LIN {X 0,Y 487.577,Z 898.273,A -85,B 0,C 180,E1 21910.239,E2 21910.239} C_VEL
LIN {X 0,Y 482.825,Z 918.479,A -85,B 0,C 180,E1 21908.672,E2 21908.672} C_VEL
LIN {X 0,Y 477.745,Z 938.393,A -85,B 0,C 180,E1 21906.843,E2 21906.843} C_VEL
LIN {X 0,Y 473.211,Z 955.74,A -85,B 0,C 180,E1 21905.007,E2 21905.007} C_VEL
LIN {X 0,Y 468.212,Z 974.396,A -85,B 0,C 180,E1 21902.704,E2 21902.704} C_VEL
LIN {X 0,Y 464.166,Z 989.477,A -85,B 0,C 180,E1 21900.556,E2 21900.556} C_VEL
LIN {X 0,Y 459.907,Z 1005.746,A -85,B 0,C 180,E1 21897.868,E2 21897.868} C_VEL
LIN {X 0,Y 456.712,Z 1018.542,A -85,B 0,C 180,E1 21895.411,E2 21895.411} C_VEL
LIN {X 0,Y 453.523,Z 1032.445,A -85,B 0,C 180,E1 21892.285,E2 21892.285} C_VEL
LIN {X 0,Y 451.526,Z 1042.299,A -85,B 0,C 180,E1 21889.67,E2 21889.67} C_VEL
LIN {X 0,Y 449.832,Z 1052.269,A -85,B 0,C 180,E1 21886.53,E2 21886.53} C_VEL
LIN {X 0,Y 448.876,Z 1059.387,A -85,B 0,C 180,E1 21883.781,E2 21883.781} C_VEL
LIN {X 0,Y 448.274,Z 1065.688,A -85,B 0,C 180,E1 21880.799,E2 21880.799} C_VEL
LIN {X 0,Y 447.995,Z 1070.282,A -85,B 0,C 180,E1 21877.825,E2 21877.825} C_VEL
LIN {X 0,Y 447.945,Z 1073.099,A -85,B 0,C 180,E1 21875.251,E2 21875.251} C_VEL
LIN {X 0,Y 447.938,Z 1075.03,A -85,B 0,C 180,E1 21872.303,E2 21872.303} C_VEL
LIN {X 0,Y 447.939,Z 1075.344,A -85,B 0,C 180,E1 21869.361,E2 21869.361} C_VEL
LIN {X 0,Y 447.943,Z 1074.469,A -85,B 0,C 180,E1 21866.801,E2 21866.801} C_VEL
LIN {X 0,Y 447.955,Z 1072.272,A -85,B 0,C 180,E1 21863.978,E2 21863.978} C_VEL
LIN {X 0,Y 448.079,Z 1068.203,A -85,B 0,C 180,E1 21860.884,E2 21860.884} C_VEL
LIN {X 0,Y 448.424,Z 1063.366,A -85,B 0,C 180,E1 21858.204,E2 21858.204} C_VEL
LIN {X 0,Y 449.173,Z 1056.41,A -85,B 0,C 180,E1 21855.167,E2 21855.167} C_VEL
LIN {X 0,Y 450.365,Z 1048.003,A -85,B 0,C 180,E1 21852.262,E2 21852.262} C_VEL
LIN {X 0,Y 452.098,Z 1038.249,A -85,B 0,C 180,E1 21849.411,E2 21849.411} C_VEL
LIN {X 0,Y 454.492,Z 1026.41,A -85,B 0,C 180,E1 21846.534,E2 21846.534} C_VEL
LIN {X 0,Y 457.338,Z 1014.003,A -85,B 0,C 180,E1 21843.931,E2 21843.931} C_VEL
LIN {X 0,Y 461.01,Z 998.825,A -85,B 0,C 180,E1 21841.217,E2 21841.217} C_VEL
LIN {X 0,Y 464.563,Z 984.836,A -85,B 0,C 180,E1 21839.042,E2 21839.042} C_VEL
LIN {X 0,Y 469.251,Z 966.475,A -85,B 0,C 180,E1 21836.577,E2 21836.577} C_VEL
LIN {X 0,Y 473.301,Z 950.565,A -85,B 0,C 180,E1 21834.731,E2 21834.731} C_VEL
LIN {X 0,Y 478.374,Z 930.215,A -85,B 0,C 180,E1 21832.688,E2 21832.688} C_VEL
LIN {X 0,Y 482.676,Z 911.955,A -85,B 0,C 180,E1 21831.121,E2 21831.121} C_VEL
LIN {X 0,Y 487.326,Z 891.147,A -85,B 0,C 180,E1 21829.572,E2 21829.572} C_VEL
LIN {X 0,Y 491.661,Z 869.604,A -85,B 0,C 180,E1 21828.238,E2 21828.238} C_VEL
LIN {X 0,Y 495.61,Z 848.055,A -85,B 0,C 180,E1 21827.107,E2 21827.107} C_VEL
LIN {X 0,Y 499.321,Z 824.384,A -85,B 0,C 180,E1 21826.103,E2 21826.103} C_VEL
LIN {X 0,Y 502.303,Z 802.272,A -85,B 0,C 180,E1 21825.352,E2 21825.352} C_VEL
LIN {X 0,Y 504.984,Z 776.643,A -85,B 0,C 180,E1 21824.697,E2 21824.697} C_VEL
LIN {X 0,Y 506.564,Z 754.118,A -85,B 0,C 180,E1 21824.276,E2 21824.276} C_VEL
LIN {X 0,Y 516.933,Z 505.006,A -85,B 0,C 180,E1 21820.505,E2 21820.505} C_VEL
LIN {X 0,Y 518.425,Z 466.807,A -85,B 0,C 180,E1 21819.907,E2 21819.907} C_VEL
LIN {X 0,Y 506.72,Z 446.358,A -85,B 0,C 180,E1 21817.91,E2 21817.91} C_VEL
LIN {X 0,Y 496.467,Z 429.865,A -85,B 0,C 180,E1 21816.04,E2 21816.04} C_VEL
LIN {X 0,Y 486.048,Z 414.014,A -85,B 0,C 180,E1 21813.99,E2 21813.99} C_VEL
LIN {X 0,Y 476.62,Z 400.744,A -85,B 0,C 180,E1 21811.986,E2 21811.986} C_VEL
LIN {X 0,Y 470.189,Z 391.86,A -85,B 0,C 180,E1 21810.512,E2 21810.512} C_VEL
LIN {X 0,Y 465.532,Z 385.893,A -85,B 0,C 180,E1 21809.392,E2 21809.392} C_VEL
LIN {X 0,Y 461.918,Z 381.059,A -85,B 0,C 180,E1 21808.474,E2 21808.474} C_VEL
LIN {X 0,Y 456.914,Z 374.765,A -85,B 0,C 180,E1 21807.147,E2 21807.147} C_VEL
LIN {X 0,Y 453.412,Z 370.552,A -85,B 0,C 180,E1 21806.171,E2 21806.171} C_VEL
LIN {X 0,Y 451.1,Z 367.867,A -85,B 0,C 180,E1 21805.504,E2 21805.504} C_VEL
LIN {X 0,Y 450.288,Z 365.126,A -85,B 0,C 180,E1 21804.741,E2 21804.741} C_VEL
LIN {X 0,Y 450.26,Z 365.145,A -85,B 0,C 180,E1 21801.142,E2 21801.142} C_VEL
LIN {X 0,Y 450.242,Z 365.132,A -85,B 0,C 180,E1 21797.446,E2 21797.446} C_VEL
LIN {X 0,Y 450.24,Z 365.115,A -85,B 0,C 180,E1 21793.746,E2 21793.746} C_VEL
LIN {X 0,Y 450.274,Z 365.11,A -85,B 0,C 180,E1 21790.233,E2 21790.233} C_VEL
LIN {X 0,Y 450.299,Z 365.136,A -85,B 0,C 180,E1 21786.502,E2 21786.502} C_VEL
LIN {X 0,Y 450.259,Z 365.128,A -85,B 0,C 180,E1 21782.8,E2 21782.8} C_VEL
LIN {X 0,Y 450.236,Z 365.107,A -85,B 0,C 180,E1 21779.237,E2 21779.237} C_VEL
LIN {X 0,Y 450.246,Z 365.129,A -85,B 0,C 180,E1 21775.542,E2 21775.542} C_VEL
LIN {X 0,Y 450.282,Z 365.135,A -85,B 0,C 180,E1 21771.958,E2 21771.958} C_VEL
LIN {X 0,Y 450.284,Z 365.106,A -85,B 0,C 180,E1 21768.212,E2 21768.212} C_VEL
LIN {X 0,Y 450.249,Z 365.117,A -85,B 0,C 180,E1 21764.676,E2 21764.676} C_VEL
LIN {X 0,Y 450.245,Z 365.146,A -85,B 0,C 180,E1 21761.081,E2 21761.081} C_VEL
LIN {X 0,Y 450.26,Z 365.134,A -85,B 0,C 180,E1 21757.407,E2 21757.407} C_VEL
LIN {X 0,Y 450.29,Z 365.115,A -85,B 0,C 180,E1 21753.775,E2 21753.775} C_VEL
LIN {X 0,Y 450.287,Z 365.336,A -85,B 0,C 180,E1 21752.375,E2 21752.375} C_VEL
LIN {X 0,Y 451.296,Z 368.138,A -85,B 0,C 180,E1 21752.02,E2 21752.02} C_VEL
LIN {X 0,Y 453.847,Z 370.847,A -85,B 0,C 180,E1 21751.296,E2 21751.296} C_VEL
LIN {X 0,Y 455.527,Z 371.957,A -85,B 0,C 180,E1 21750.855,E2 21750.855} C_VEL
LIN {X 0,Y 457.684,Z 375.518,A -85,B 0,C 180,E1 21750.233,E2 21750.233} C_VEL
LIN {X 0,Y 460.657,Z 378.21,A -85,B 0,C 180,E1 21749.475,E2 21749.475} C_VEL
LIN {X 0,Y 463.451,Z 382.175,A -85,B 0,C 180,E1 21748.743,E2 21748.743} C_VEL
LIN {X 0,Y 465.734,Z 384.434,A -85,B 0,C 180,E1 21748.192,E2 21748.192} C_VEL
LIN {X 0,Y 469.137,Z 388.783,A -85,B 0,C 180,E1 21747.369,E2 21747.369} C_VEL
LIN {X 0,Y 470.884,Z 390.867,A -85,B 0,C 180,E1 21746.962,E2 21746.962} C_VEL
LIN {X 0,Y 476.097,Z 397.437,A -85,B 0,C 180,E1 21745.783,E2 21745.783} C_VEL
LIN {X 0,Y 480.36,Z 402.894,A -85,B 0,C 180,E1 21744.862,E2 21744.862} C_VEL
LIN {X 0,Y 487.396,Z 412.001,A -85,B 0,C 180,E1 21743.419,E2 21743.419} C_VEL
LIN {X 0,Y 499.444,Z 428.57,A -85,B 0,C 180,E1 21741.124,E2 21741.124} C_VEL
LIN {X 0,Y 511.635,Z 446.615,A -85,B 0,C 180,E1 21738.992,E2 21738.992} C_VEL
LIN {X 0,Y 518.739,Z 458.868,A -85,B 0,C 180,E1 21737.8,E2 21737.8} C_VEL
LIN {X 0,Y 508.149,Z 709.985,A -85,B 0,C 180,E1 21734.008,E2 21734.008} C_VEL
LIN {X 0,Y 506.28,Z 748.548,A -85,B 0,C 180,E1 21733.388,E2 21733.388} C_VEL
LIN {X 0,Y 504.192,Z 772.045,A -85,B 0,C 180,E1 21732.838,E2 21732.838} C_VEL
LIN {X 0,Y 501.494,Z 795.854,A -85,B 0,C 180,E1 21732.105,E2 21732.105} C_VEL
LIN {X 0,Y 498.135,Z 818.964,A -85,B 0,C 180,E1 21731.177,E2 21731.177} C_VEL
LIN {X 0,Y 494.465,Z 841.146,A -85,B 0,C 180,E1 21730.095,E2 21730.095} C_VEL
LIN {X 0,Y 490.296,Z 862.557,A -85,B 0,C 180,E1 21728.827,E2 21728.827} C_VEL
LIN {X 0,Y 486.249,Z 881.746,A -85,B 0,C 180,E1 21727.494,E2 21727.494} C_VEL
LIN {X 0,Y 481.239,Z 903.419,A -85,B 0,C 180,E1 21725.721,E2 21725.721} C_VEL
LIN {X 0,Y 477.113,Z 920.181,A -85,B 0,C 180,E1 21724.126,E2 21724.126} C_VEL
LIN {X 0,Y 472.225,Z 939.257,A -85,B 0,C 180,E1 21722.033,E2 21722.033} C_VEL
LIN {X 0,Y 468.005,Z 955.157,A -85,B 0,C 180,E1 21719.996,E2 21719.996} C_VEL
LIN {X 0,Y 463.735,Z 971.472,A -85,B 0,C 180,E1 21717.602,E2 21717.602} C_VEL
LIN {X 0,Y 459.89,Z 986.038,A -85,B 0,C 180,E1 21715.085,E2 21715.085} C_VEL
LIN {X 0,Y 456.552,Z 999.545,A -85,B 0,C 180,E1 21712.4,E2 21712.4} C_VEL
LIN {X 0,Y 453.842,Z 1010.974,A -85,B 0,C 180,E1 21709.699,E2 21709.699} C_VEL
LIN {X 0,Y 451.777,Z 1020.868,A -85,B 0,C 180,E1 21706.987,E2 21706.987} C_VEL
LIN {X 0,Y 451.27,Z 1023.48,A -85,B 0,C 180,E1 21706.176,E2 21706.176} C_VEL
LIN {X 0,Y 449.761,Z 1026.387,A -85,B 0,C 180,E1 21705.278,E2 21705.278} C_VEL
LIN {X 0,Y 442.431,Z 1033.675,A -85,B 0,C 180,E1 21702.889,E2 21702.889} C_VEL
LIN {X 0,Y 441.394,Z 1035.6,A -85,B 0,C 180,E1 21702.074,E2 21702.074} C_VEL
LIN {X 0,Y 440.648,Z 1041.384,A -85,B 0,C 180,E1 21699.271,E2 21699.271} C_VEL
LIN {X 0,Y 440.168,Z 1046.479,A -85,B 0,C 180,E1 21695.998,E2 21695.998} C_VEL
LIN {X 0,Y 440.009,Z 1049.381,A -85,B 0,C 180,E1 21693.257,E2 21693.257} C_VEL
LIN {X 0,Y 439.954,Z 1051.147,A -85,B 0,C 180,E1 21690.521,E2 21690.521} C_VEL
LIN {X 0,Y 439.94,Z 1051.693,A -85,B 0,C 180,E1 21687.395,E2 21687.395} C_VEL
LIN {X 0,Y 439.969,Z 1050.878,A -85,B 0,C 180,E1 21684.654,E2 21684.654} C_VEL
LIN {X 0,Y 440.043,Z 1049.04,A -85,B 0,C 180,E1 21682.033,E2 21682.033} C_VEL
LIN {X 0,Y 440.31,Z 1045.196,A -85,B 0,C 180,E1 21678.738,E2 21678.738} C_VEL
LIN {X 0,Y 440.816,Z 1040.543,A -85,B 0,C 180,E1 21675.954,E2 21675.954} C_VEL
LIN {X 0,Y 441.744,Z 1034.349,A -85,B 0,C 180,E1 21673.023,E2 21673.023} C_VEL
LIN {X 0,Y 443.258,Z 1026.119,A -85,B 0,C 180,E1 21669.948,E2 21669.948} C_VEL
LIN {X 0,Y 445.115,Z 1017.55,A -85,B 0,C 180,E1 21667.271,E2 21667.271} C_VEL
LIN {X 0,Y 448.164,Z 1005.199,A -85,B 0,C 180,E1 21664.044,E2 21664.044} C_VEL
LIN {X 0,Y 451.208,Z 993.916,A -85,B 0,C 180,E1 21661.546,E2 21661.546} C_VEL
LIN {X 0,Y 455.553,Z 978.507,A -85,B 0,C 180,E1 21658.629,E2 21658.629} C_VEL
LIN {X 0,Y 459.705,Z 964.184,A -85,B 0,C 180,E1 21656.314,E2 21656.314} C_VEL
LIN {X 0,Y 465.039,Z 945.702,A -85,B 0,C 180,E1 21653.752,E2 21653.752} C_VEL
LIN {X 0,Y 469.537,Z 929.823,A -85,B 0,C 180,E1 21651.862,E2 21651.862} C_VEL
LIN {X 0,Y 475.157,Z 909.241,A -85,B 0,C 180,E1 21649.757,E2 21649.757} C_VEL
LIN {X 0,Y 479.806,Z 891.095,A -85,B 0,C 180,E1 21648.175,E2 21648.175} C_VEL
LIN {X 0,Y 484.96,Z 869.463,A -85,B 0,C 180,E1 21646.559,E2 21646.559} C_VEL
LIN {X 0,Y 489.182,Z 849.717,A -85,B 0,C 180,E1 21645.321,E2 21645.321} C_VEL
LIN {X 0,Y 493.411,Z 827.942,A -85,B 0,C 180,E1 21644.162,E2 21644.162} C_VEL
LIN {X 0,Y 497.108,Z 805.082,A -85,B 0,C 180,E1 21643.178,E2 21643.178} C_VEL
LIN {X 0,Y 499.914,Z 784.791,A -85,B 0,C 180,E1 21642.467,E2 21642.467} C_VEL
LIN {X 0,Y 502.662,Z 759.493,A -85,B 0,C 180,E1 21641.784,E2 21641.784} C_VEL
LIN {X 0,Y 504.273,Z 737.798,A -85,B 0,C 180,E1 21641.358,E2 21641.358} C_VEL
LIN {X 0,Y 515.677,Z 490.781,A -85,B 0,C 180,E1 21637.581,E2 21637.581} C_VEL
LIN {X 0,Y 516.812,Z 463.843,A -85,B 0,C 180,E1 21637.148,E2 21637.148} C_VEL
LIN {X 0,Y 508.755,Z 450.942,A -85,B 0,C 180,E1 21635.678,E2 21635.678} C_VEL
LIN {X 0,Y 496.361,Z 433.111,A -85,B 0,C 180,E1 21633.26,E2 21633.26} C_VEL
LIN {X 0,Y 485.835,Z 418.911,A -85,B 0,C 180,E1 21631,E2 21631} C_VEL
LIN {X 0,Y 476.902,Z 407.617,A -85,B 0,C 180,E1 21628.9,E2 21628.9} C_VEL
LIN {X 0,Y 472.696,Z 402.404,A -85,B 0,C 180,E1 21627.837,E2 21627.837} C_VEL
LIN {X 0,Y 468.223,Z 396.919,A -85,B 0,C 180,E1 21626.645,E2 21626.645} C_VEL
LIN {X 0,Y 464.612,Z 392.56,A -85,B 0,C 180,E1 21625.631,E2 21625.631} C_VEL
LIN {X 0,Y 463.434,Z 391.165,A -85,B 0,C 180,E1 21625.29,E2 21625.29} C_VEL
LIN {X 0,Y 460.056,Z 387.445,A -85,B 0,C 180,E1 21624.288,E2 21624.288} C_VEL
LIN {X 0,Y 458.701,Z 385.415,A -85,B 0,C 180,E1 21623.851,E2 21623.851} C_VEL
LIN {X 0,Y 455.354,Z 382.348,A -85,B 0,C 180,E1 21622.803,E2 21622.803} C_VEL
LIN {X 0,Y 453.524,Z 379.251,A -85,B 0,C 180,E1 21622.148,E2 21622.148} C_VEL
LIN {X 0,Y 450.179,Z 376.741,A -85,B 0,C 180,E1 21621.021,E2 21621.021} C_VEL
LIN {X 0,Y 448.267,Z 373.433,A -85,B 0,C 180,E1 21620.261,E2 21620.261} C_VEL
LIN {X 0,Y 447.894,Z 372.768,A -85,B 0,C 180,E1 21620.108,E2 21620.108} C_VEL
LIN {X 0,Y 444.635,Z 370.837,A -85,B 0,C 180,E1 21618.895,E2 21618.895} C_VEL
LIN {X 0,Y 442.875,Z 368.133,A -85,B 0,C 180,E1 21618.12,E2 21618.12} C_VEL
LIN {X 0,Y 442.338,Z 366.106,A -85,B 0,C 180,E1 21617.768,E2 21617.768} C_VEL
LIN {X 0,Y 442.359,Z 366.102,A -85,B 0,C 180,E1 21613.996,E2 21613.996} C_VEL
LIN {X 0,Y 442.321,Z 366.108,A -85,B 0,C 180,E1 21610.287,E2 21610.287} C_VEL
LIN {X 0,Y 442.3,Z 366.118,A -85,B 0,C 180,E1 21606.751,E2 21606.751} C_VEL
LIN {X 0,Y 442.306,Z 366.128,A -85,B 0,C 180,E1 21602.98,E2 21602.98} C_VEL
LIN {X 0,Y 442.335,Z 366.134,A -85,B 0,C 180,E1 21599.352,E2 21599.352} C_VEL
LIN {X 0,Y 442.347,Z 366.12,A -85,B 0,C 180,E1 21595.592,E2 21595.592} C_VEL
LIN {X 0,Y 442.325,Z 366.11,A -85,B 0,C 180,E1 21591.937,E2 21591.937} C_VEL
LIN {X 0,Y 442.302,Z 366.107,A -85,B 0,C 180,E1 21588.261,E2 21588.261} C_VEL
LIN {X 0,Y 442.299,Z 366.106,A -85,B 0,C 180,E1 21584.528,E2 21584.528} C_VEL
LIN {X 0,Y 442.314,Z 366.105,A -85,B 0,C 180,E1 21580.866,E2 21580.866} C_VEL
LIN {X 0,Y 442.322,Z 366.277,A -85,B 0,C 180,E1 21580.516,E2 21580.516} C_VEL
LIN {X 0,Y 443.214,Z 368.939,A -85,B 0,C 180,E1 21580.049,E2 21580.049} C_VEL
LIN {X 0,Y 445.677,Z 371.68,A -85,B 0,C 180,E1 21579.032,E2 21579.032} C_VEL
LIN {X 0,Y 448.061,Z 373.157,A -85,B 0,C 180,E1 21578.154,E2 21578.154} C_VEL
LIN {X 0,Y 450.632,Z 377.217,A -85,B 0,C 180,E1 21577.151,E2 21577.151} C_VEL
LIN {X 0,Y 453.238,Z 379.579,A -85,B 0,C 180,E1 21576.258,E2 21576.258} C_VEL
LIN {X 0,Y 458.645,Z 386.423,A -85,B 0,C 180,E1 21574.462,E2 21574.462} C_VEL
LIN {X 0,Y 461.948,Z 390.347,A -85,B 0,C 180,E1 21573.45,E2 21573.45} C_VEL
LIN {X 0,Y 467.029,Z 396.989,A -85,B 0,C 180,E1 21571.969,E2 21571.969} C_VEL
LIN {X 0,Y 474.172,Z 406.465,A -85,B 0,C 180,E1 21570.05,E2 21570.05} C_VEL
LIN {X 0,Y 482.866,Z 418.454,A -85,B 0,C 180,E1 21567.917,E2 21567.917} C_VEL
LIN {X 0,Y 490.981,Z 430.365,A -85,B 0,C 180,E1 21566.082,E2 21566.082} C_VEL
LIN {X 0,Y 498.672,Z 442.104,A -85,B 0,C 180,E1 21564.463,E2 21564.463} C_VEL
LIN {X 0,Y 508.434,Z 457.967,A -85,B 0,C 180,E1 21562.542,E2 21562.542} C_VEL
LIN {X 0,Y 516.756,Z 472.571,A -85,B 0,C 180,E1 21561.002,E2 21561.002} C_VEL
LIN {X 0,Y 505.459,Z 719.112,A -85,B 0,C 180,E1 21557.239,E2 21557.239} C_VEL
LIN {X 0,Y 503.141,Z 765.997,A -85,B 0,C 180,E1 21556.494,E2 21556.494} C_VEL
LIN {X 0,Y 500.731,Z 790.293,A -85,B 0,C 180,E1 21555.946,E2 21555.946} C_VEL
LIN {X 0,Y 498.012,Z 811.651,A -85,B 0,C 180,E1 21555.318,E2 21555.318} C_VEL
LIN {X 0,Y 494.284,Z 835.385,A -85,B 0,C 180,E1 21554.421,E2 21554.421} C_VEL
LIN {X 0,Y 490.661,Z 855.328,A -85,B 0,C 180,E1 21553.492,E2 21553.492} C_VEL
LIN {X 0,Y 485.976,Z 878.276,A -85,B 0,C 180,E1 21552.209,E2 21552.209} C_VEL
LIN {X 0,Y 481.392,Z 898.253,A -85,B 0,C 180,E1 21550.865,E2 21550.865} C_VEL
LIN {X 0,Y 476.571,Z 918.04,A -85,B 0,C 180,E1 21549.318,E2 21549.318} C_VEL
LIN {X 0,Y 471.365,Z 937.738,A -85,B 0,C 180,E1 21547.5,E2 21547.5} C_VEL
LIN {X 0,Y 466.637,Z 955.097,A -85,B 0,C 180,E1 21545.65,E2 21545.65} C_VEL
LIN {X 0,Y 461.543,Z 973.356,A -85,B 0,C 180,E1 21543.385,E2 21543.385} C_VEL
LIN {X 0,Y 457.296,Z 988.506,A -85,B 0,C 180,E1 21541.212,E2 21541.212} C_VEL
LIN {X 0,Y 452.79,Z 1004.901,A -85,B 0,C 180,E1 21538.489,E2 21538.489} C_VEL
LIN {X 0,Y 449.393,Z 1017.799,A -85,B 0,C 180,E1 21535.987,E2 21535.987} C_VEL
LIN {X 0,Y 446.251,Z 1030.721,A -85,B 0,C 180,E1 21533.086,E2 21533.086} C_VEL
LIN {X 0,Y 443.949,Z 1041.201,A -85,B 0,C 180,E1 21530.295,E2 21530.295} C_VEL
LIN {X 0,Y 442.159,Z 1051.012,A -85,B 0,C 180,E1 21527.232,E2 21527.232} C_VEL
LIN {X 0,Y 440.987,Z 1058.875,A -85,B 0,C 180,E1 21524.175,E2 21524.175} C_VEL
LIN {X 0,Y 440.343,Z 1064.981,A -85,B 0,C 180,E1 21521.261,E2 21521.261} C_VEL
LIN {X 0,Y 440.015,Z 1069.92,A -85,B 0,C 180,E1 21518.099,E2 21518.099} C_VEL
LIN {X 0,Y 439.947,Z 1072.8,A -85,B 0,C 180,E1 21515.455,E2 21515.455} C_VEL
LIN {X 0,Y 439.94,Z 1074.616,A -85,B 0,C 180,E1 21512.736,E2 21512.736} C_VEL
LIN {X 0,Y 439.941,Z 1075.173,A -85,B 0,C 180,E1 21509.609,E2 21509.609} C_VEL
LIN {X 0,Y 439.945,Z 1074.317,A -85,B 0,C 180,E1 21506.873,E2 21506.873} C_VEL
LIN {X 0,Y 439.954,Z 1072.278,A -85,B 0,C 180,E1 21504.13,E2 21504.13} C_VEL
LIN {X 0,Y 440.072,Z 1068.387,A -85,B 0,C 180,E1 21500.98,E2 21500.98} C_VEL
LIN {X 0,Y 440.422,Z 1063.558,A -85,B 0,C 180,E1 21498.21,E2 21498.21} C_VEL
LIN {X 0,Y 441.131,Z 1057.143,A -85,B 0,C 180,E1 21495.294,E2 21495.294} C_VEL
LIN {X 0,Y 442.378,Z 1048.656,A -85,B 0,C 180,E1 21492.234,E2 21492.234} C_VEL
LIN {X 0,Y 444.002,Z 1039.698,A -85,B 0,C 180,E1 21489.527,E2 21489.527} C_VEL
LIN {X 0,Y 446.636,Z 1027.29,A -85,B 0,C 180,E1 21486.376,E2 21486.376} C_VEL
LIN {X 0,Y 449.397,Z 1015.646,A -85,B 0,C 180,E1 21483.862,E2 21483.862} C_VEL
LIN {X 0,Y 453.148,Z 1000.861,A -85,B 0,C 180,E1 21481.103,E2 21481.103} C_VEL
LIN {X 0,Y 456.994,Z 986.23,A -85,B 0,C 180,E1 21478.765,E2 21478.765} C_VEL
LIN {X 0,Y 461.561,Z 969.219,A -85,B 0,C 180,E1 21476.393,E2 21476.393} C_VEL
LIN {X 0,Y 466.175,Z 951.698,A -85,B 0,C 180,E1 21474.309,E2 21474.309} C_VEL
LIN {X 0,Y 471.19,Z 932.534,A -85,B 0,C 180,E1 21472.327,E2 21472.327} C_VEL
LIN {X 0,Y 475.946,Z 913.043,A -85,B 0,C 180,E1 21470.62,E2 21470.62} C_VEL
LIN {X 0,Y 480.325,Z 894.144,A -85,B 0,C 180,E1 21469.182,E2 21469.182} C_VEL
LIN {X 0,Y 485.174,Z 871.29,A -85,B 0,C 180,E1 21467.72,E2 21467.72} C_VEL
LIN {X 0,Y 489.097,Z 850.681,A -85,B 0,C 180,E1 21466.614,E2 21466.614} C_VEL
LIN {X 0,Y 493.184,Z 826.007,A -85,B 0,C 180,E1 21465.533,E2 21465.533} C_VEL
LIN {X 0,Y 496.178,Z 804.692,A -85,B 0,C 180,E1 21464.793,E2 21464.793} C_VEL
LIN {X 0,Y 498.987,Z 779.88,A -85,B 0,C 180,E1 21464.126,E2 21464.126} C_VEL
LIN {X 0,Y 500.74,Z 756.733,A -85,B 0,C 180,E1 21463.676,E2 21463.676} C_VEL
LIN {X 0,Y 511.241,Z 514.011,A -85,B 0,C 180,E1 21459.97,E2 21459.97} C_VEL
LIN {X 0,Y 513.043,Z 470.309,A -85,B 0,C 180,E1 21459.284,E2 21459.284} C_VEL
LIN {X 0,Y 502.048,Z 450.985,A -85,B 0,C 180,E1 21457.351,E2 21457.351} C_VEL
LIN {X 0,Y 490.607,Z 432.404,A -85,B 0,C 180,E1 21455.188,E2 21455.188} C_VEL
LIN {X 0,Y 478.766,Z 414.63,A -85,B 0,C 180,E1 21452.746,E2 21452.746} C_VEL
LIN {X 0,Y 467.489,Z 398.866,A -85,B 0,C 180,E1 21450.174,E2 21450.174} C_VEL
LIN {X 0,Y 458.988,Z 387.726,A -85,B 0,C 180,E1 21448.035,E2 21448.035} C_VEL
LIN {X 0,Y 454.272,Z 381.695,A -85,B 0,C 180,E1 21446.752,E2 21446.752} C_VEL
LIN {X 0,Y 451.019,Z 377.76,A -85,B 0,C 180,E1 21445.826,E2 21445.826} C_VEL
LIN {X 0,Y 448.461,Z 374.594,A -85,B 0,C 180,E1 21445.064,E2 21445.064} C_VEL
LIN {X 0,Y 446.748,Z 372.301,A -85,B 0,C 180,E1 21444.531,E2 21444.531} C_VEL
LIN {X 0,Y 443.911,Z 370.013,A -85,B 0,C 180,E1 21443.672,E2 21443.672} C_VEL
LIN {X 0,Y 442.519,Z 367.142,A -85,B 0,C 180,E1 21443.169,E2 21443.169} C_VEL
LIN {X 0,Y 442.344,Z 366.098,A -85,B 0,C 180,E1 21442.88,E2 21442.88} C_VEL
LIN {X 0,Y 442.308,Z 366.102,A -85,B 0,C 180,E1 21439.272,E2 21439.272} C_VEL
LIN {X 0,Y 442.3,Z 366.115,A -85,B 0,C 180,E1 21435.606,E2 21435.606} C_VEL
LIN {X 0,Y 442.32,Z 366.136,A -85,B 0,C 180,E1 21432.004,E2 21432.004} C_VEL
LIN {X 0,Y 442.348,Z 366.102,A -85,B 0,C 180,E1 21428.318,E2 21428.318} C_VEL
LIN {X 0,Y 442.33,Z 366.094,A -85,B 0,C 180,E1 21424.668,E2 21424.668} C_VEL
LIN {X 0,Y 442.307,Z 366.123,A -85,B 0,C 180,E1 21421.036,E2 21421.036} C_VEL
LIN {X 0,Y 442.302,Z 366.125,A -85,B 0,C 180,E1 21417.279,E2 21417.279} C_VEL
LIN {X 0,Y 442.305,Z 366.098,A -85,B 0,C 180,E1 21413.51,E2 21413.51} C_VEL
LIN {X 0,Y 442.341,Z 366.102,A -85,B 0,C 180,E1 21409.976,E2 21409.976} C_VEL
LIN {X 0,Y 442.36,Z 366.13,A -85,B 0,C 180,E1 21406.137,E2 21406.137} C_VEL
LIN {X 0,Y 442.33,Z 366.113,A -85,B 0,C 180,E1 21402.368,E2 21402.368} C_VEL
LIN {X 0,Y 442.304,Z 366.101,A -85,B 0,C 180,E1 21398.795,E2 21398.795} C_VEL
LIN {X 0,Y 442.305,Z 366.104,A -85,B 0,C 180,E1 21395.028,E2 21395.028} C_VEL
LIN {X 0,Y 442.339,Z 366.294,A -85,B 0,C 180,E1 21394.499,E2 21394.499} C_VEL
LIN {X 0,Y 443.294,Z 369.02,A -85,B 0,C 180,E1 21394.122,E2 21394.122} C_VEL
LIN {X 0,Y 445.743,Z 371.73,A -85,B 0,C 180,E1 21393.343,E2 21393.343} C_VEL
LIN {X 0,Y 447.768,Z 373.027,A -85,B 0,C 180,E1 21392.756,E2 21392.756} C_VEL
LIN {X 0,Y 449.926,Z 376.626,A -85,B 0,C 180,E1 21392.072,E2 21392.072} C_VEL
LIN {X 0,Y 453.113,Z 379.439,A -85,B 0,C 180,E1 21391.185,E2 21391.185} C_VEL
LIN {X 0,Y 455.896,Z 383.357,A -85,B 0,C 180,E1 21390.394,E2 21390.394} C_VEL
LIN {X 0,Y 458.238,Z 385.663,A -85,B 0,C 180,E1 21389.782,E2 21389.782} C_VEL
LIN {X 0,Y 461.633,Z 389.986,A -85,B 0,C 180,E1 21388.896,E2 21388.896} C_VEL
LIN {X 0,Y 463.272,Z 391.839,A -85,B 0,C 180,E1 21388.489,E2 21388.489} C_VEL
LIN {X 0,Y 467.173,Z 396.479,A -85,B 0,C 180,E1 21387.542,E2 21387.542} C_VEL
LIN {X 0,Y 476.963,Z 409.138,A -85,B 0,C 180,E1 21385.308,E2 21385.308} C_VEL
LIN {X 0,Y 484.786,Z 419.482,A -85,B 0,C 180,E1 21383.668,E2 21383.668} C_VEL
LIN {X 0,Y 496.615,Z 435.891,A -85,B 0,C 180,E1 21381.379,E2 21381.379} C_VEL
LIN {X 0,Y 508.771,Z 454.299,A -85,B 0,C 180,E1 21379.215,E2 21379.215} C_VEL
LIN {X 0,Y 513.368,Z 462.385,A -85,B 0,C 180,E1 21378.424,E2 21378.424} C_VEL
LIN {X 0,Y 502.343,Z 714.904,A -85,B 0,C 180,E1 21374.583,E2 21374.583} C_VEL
LIN {X 0,Y 500.516,Z 749.833,A -85,B 0,C 180,E1 21374.008,E2 21374.008} C_VEL
LIN {X 0,Y 498.414,Z 772.695,A -85,B 0,C 180,E1 21373.466,E2 21373.466} C_VEL
LIN {X 0,Y 495.629,Z 796.424,A -85,B 0,C 180,E1 21372.728,E2 21372.728} C_VEL
LIN {X 0,Y 492.352,Z 818.328,A -85,B 0,C 180,E1 21371.846,E2 21371.846} C_VEL
LIN {X 0,Y 488.749,Z 839.499,A -85,B 0,C 180,E1 21370.816,E2 21370.816} C_VEL
LIN {X 0,Y 484.276,Z 862.069,A -85,B 0,C 180,E1 21369.489,E2 21369.489} C_VEL
LIN {X 0,Y 480.234,Z 880.63,A -85,B 0,C 180,E1 21368.198,E2 21368.198} C_VEL
LIN {X 0,Y 475.211,Z 901.882,A -85,B 0,C 180,E1 21366.47,E2 21366.47} C_VEL
LIN {X 0,Y 470.686,Z 919.635,A -85,B 0,C 180,E1 21364.777,E2 21364.777} C_VEL
LIN {X 0,Y 465.808,Z 938.147,A -85,B 0,C 180,E1 21362.747,E2 21362.747} C_VEL
LIN {X 0,Y 461.166,Z 954.845,A -85,B 0,C 180,E1 21360.597,E2 21360.597} C_VEL
LIN {X 0,Y 456.779,Z 970.943,A -85,B 0,C 180,E1 21358.218,E2 21358.218} C_VEL
LIN {X 0,Y 452.707,Z 985.688,A -85,B 0,C 180,E1 21355.652,E2 21355.652} C_VEL
LIN {X 0,Y 449.323,Z 998.642,A -85,B 0,C 180,E1 21353.058,E2 21353.058} C_VEL
LIN {X 0,Y 446.265,Z 1010.913,A -85,B 0,C 180,E1 21350.148,E2 21350.148} C_VEL
LIN {X 0,Y 444.102,Z 1020.716,A -85,B 0,C 180,E1 21347.424,E2 21347.424} C_VEL
LIN {X 0,Y 442.278,Z 1030.14,A -85,B 0,C 180,E1 21344.266,E2 21344.266} C_VEL
LIN {X 0,Y 441.394,Z 1035.6,A -85,B 0,C 180,E1 21342.074,E2 21342.074} C_VEL
LIN {X 0,Y 440.111,Z 1037.86,A -85,B 0,C 180,E1 21341.12,E2 21341.12} C_VEL
LIN {X 0,Y 433.155,Z 1043.266,A -85,B 0,C 180,E1 21338.498,E2 21338.498} C_VEL
LIN {X 0,Y 432.383,Z 1044.478,A -85,B 0,C 180,E1 21337.711,E2 21337.711} C_VEL
LIN {X 0,Y 432.089,Z 1048.284,A -85,B 0,C 180,E1 21334.779,E2 21334.779} C_VEL
LIN {X 0,Y 431.976,Z 1050.837,A -85,B 0,C 180,E1 21331.592,E2 21331.592} C_VEL
LIN {X 0,Y 431.951,Z 1051.8,A -85,B 0,C 180,E1 21328.939,E2 21328.939} C_VEL
LIN {X 0,Y 431.954,Z 1051.698,A -85,B 0,C 180,E1 21326.103,E2 21326.103} C_VEL
LIN {X 0,Y 432.022,Z 1050.014,A -85,B 0,C 180,E1 21322.82,E2 21322.82} C_VEL
LIN {X 0,Y 432.173,Z 1047.424,A -85,B 0,C 180,E1 21320.142,E2 21320.142} C_VEL
LIN {X 0,Y 432.574,Z 1043.346,A -85,B 0,C 180,E1 21317.179,E2 21317.179} C_VEL
LIN {X 0,Y 433.432,Z 1037.204,A -85,B 0,C 180,E1 21313.929,E2 21313.929} C_VEL
LIN {X 0,Y 434.663,Z 1030.406,A -85,B 0,C 180,E1 21311.074,E2 21311.074} C_VEL
LIN {X 0,Y 436.848,Z 1020.417,A -85,B 0,C 180,E1 21307.669,E2 21307.669} C_VEL
LIN {X 0,Y 439.249,Z 1010.8,A -85,B 0,C 180,E1 21304.95,E2 21304.95} C_VEL
LIN {X 0,Y 442.83,Z 997.813,A -85,B 0,C 180,E1 21301.841,E2 21301.841} C_VEL
LIN {X 0,Y 446.49,Z 985.27,A -85,B 0,C 180,E1 21299.297,E2 21299.297} C_VEL
LIN {X 0,Y 451.054,Z 970.157,A -85,B 0,C 180,E1 21296.649,E2 21296.649} C_VEL
LIN {X 0,Y 455.508,Z 955.338,A -85,B 0,C 180,E1 21294.43,E2 21294.43} C_VEL
LIN {X 0,Y 460.715,Z 938.153,A -85,B 0,C 180,E1 21292.185,E2 21292.185} C_VEL
LIN {X 0,Y 465.91,Z 919.972,A -85,B 0,C 180,E1 21290.171,E2 21290.171} C_VEL
LIN {X 0,Y 470.913,Z 901.887,A -85,B 0,C 180,E1 21288.43,E2 21288.43} C_VEL
LIN {X 0,Y 476.312,Z 880.73,A -85,B 0,C 180,E1 21286.703,E2 21286.703} C_VEL
LIN {X 0,Y 480.673,Z 862.161,A -85,B 0,C 180,E1 21285.407,E2 21285.407} C_VEL
LIN {X 0,Y 485.784,Z 837.994,A -85,B 0,C 180,E1 21283.997,E2 21283.997} C_VEL
LIN {X 0,Y 489.516,Z 817.506,A -85,B 0,C 180,E1 21283.008,E2 21283.008} C_VEL
LIN {X 0,Y 493.406,Z 792.396,A -85,B 0,C 180,E1 21282.031,E2 21282.031} C_VEL
LIN {X 0,Y 496.099,Z 770.51,A -85,B 0,C 180,E1 21281.372,E2 21281.372} C_VEL
LIN {X 0,Y 498.452,Z 745.206,A -85,B 0,C 180,E1 21280.804,E2 21280.804} C_VEL
LIN {X 0,Y 501.921,Z 674.53,A -85,B 0,C 180,E1 21279.695,E2 21279.695} C_VEL
LIN {X 0,Y 511.78,Z 467.818,A -85,B 0,C 180,E1 21276.514,E2 21276.514} C_VEL
LIN {X 0,Y 504.78,Z 456.576,A -85,B 0,C 180,E1 21275.2,E2 21275.2} C_VEL
LIN {X 0,Y 492.925,Z 439.35,A -85,B 0,C 180,E1 21272.828,E2 21272.828} C_VEL
LIN {X 0,Y 482.888,Z 425.653,A -85,B 0,C 180,E1 21270.623,E2 21270.623} C_VEL
LIN {X 0,Y 474.182,Z 414.504,A -85,B 0,C 180,E1 21268.53,E2 21268.53} C_VEL
LIN {X 0,Y 470.031,Z 409.325,A -85,B 0,C 180,E1 21267.458,E2 21267.458} C_VEL
LIN {X 0,Y 465.619,Z 403.891,A -85,B 0,C 180,E1 21266.256,E2 21266.256} C_VEL
LIN {X 0,Y 461.89,Z 399.125,A -85,B 0,C 180,E1 21265.175,E2 21265.175} C_VEL
LIN {X 0,Y 457.865,Z 394.726,A -85,B 0,C 180,E1 21263.966,E2 21263.966} C_VEL
LIN {X 0,Y 456.425,Z 392.715,A -85,B 0,C 180,E1 21263.498,E2 21263.498} C_VEL
LIN {X 0,Y 452.979,Z 389.244,A -85,B 0,C 180,E1 21262.382,E2 21262.382} C_VEL
LIN {X 0,Y 451.321,Z 386.663,A -85,B 0,C 180,E1 21261.783,E2 21261.783} C_VEL
LIN {X 0,Y 447.983,Z 383.799,A -85,B 0,C 180,E1 21260.616,E2 21260.616} C_VEL
LIN {X 0,Y 445.946,Z 380.402,A -85,B 0,C 180,E1 21259.79,E2 21259.79} C_VEL
LIN {X 0,Y 442.622,Z 378.058,A -85,B 0,C 180,E1 21258.505,E2 21258.505} C_VEL
LIN {X 0,Y 440.723,Z 374.852,A -85,B 0,C 180,E1 21257.631,E2 21257.631} C_VEL
LIN {X 0,Y 440.365,Z 373.869,A -85,B 0,C 180,E1 21257.441,E2 21257.441} C_VEL
LIN {X 0,Y 437.089,Z 372.153,A -85,B 0,C 180,E1 21256.001,E2 21256.001} C_VEL
LIN {X 0,Y 435.021,Z 369.435,A -85,B 0,C 180,E1 21254.918,E2 21254.918} C_VEL
LIN {X 0,Y 434.375,Z 367.098,A -85,B 0,C 180,E1 21254.463,E2 21254.463} C_VEL
LIN {X 0,Y 434.364,Z 367.103,A -85,B 0,C 180,E1 21250.746,E2 21250.746} C_VEL
LIN {X 0,Y 434.366,Z 367.111,A -85,B 0,C 180,E1 21247.008,E2 21247.008} C_VEL
LIN {X 0,Y 434.383,Z 367.122,A -85,B 0,C 180,E1 21243.299,E2 21243.299} C_VEL
LIN {X 0,Y 434.418,Z 367.114,A -85,B 0,C 180,E1 21239.604,E2 21239.604} C_VEL
LIN {X 0,Y 434.401,Z 367.104,A -85,B 0,C 180,E1 21235.776,E2 21235.776} C_VEL
LIN {X 0,Y 434.377,Z 367.098,A -85,B 0,C 180,E1 21232.061,E2 21232.061} C_VEL
LIN {X 0,Y 434.362,Z 367.095,A -85,B 0,C 180,E1 21228.312,E2 21228.312} C_VEL
LIN {X 0,Y 434.36,Z 367.094,A -85,B 0,C 180,E1 21224.512,E2 21224.512} C_VEL
LIN {X 0,Y 434.417,Z 367.337,A -85,B 0,C 180,E1 21223.829,E2 21223.829} C_VEL
LIN {X 0,Y 435.494,Z 370.263,A -85,B 0,C 180,E1 21223.15,E2 21223.15} C_VEL
LIN {X 0,Y 437.713,Z 372.671,A -85,B 0,C 180,E1 21222.038,E2 21222.038} C_VEL
LIN {X 0,Y 440.378,Z 374.005,A -85,B 0,C 180,E1 21220.881,E2 21220.881} C_VEL
LIN {X 0,Y 442.007,Z 377.269,A -85,B 0,C 180,E1 21220.095,E2 21220.095} C_VEL
LIN {X 0,Y 445.233,Z 380.091,A -85,B 0,C 180,E1 21218.803,E2 21218.803} C_VEL
LIN {X 0,Y 446.288,Z 380.829,A -85,B 0,C 180,E1 21218.409,E2 21218.409} C_VEL
LIN {X 0,Y 448.678,Z 384.586,A -85,B 0,C 180,E1 21217.461,E2 21217.461} C_VEL
LIN {X 0,Y 451.531,Z 387.353,A -85,B 0,C 180,E1 21216.46,E2 21216.46} C_VEL
LIN {X 0,Y 459.737,Z 397.67,A -85,B 0,C 180,E1 21213.765,E2 21213.765} C_VEL
LIN {X 0,Y 464.655,Z 404.165,A -85,B 0,C 180,E1 21212.302,E2 21212.302} C_VEL
LIN {X 0,Y 471.602,Z 413.51,A -85,B 0,C 180,E1 21210.396,E2 21210.396} C_VEL
LIN {X 0,Y 481.089,Z 426.79,A -85,B 0,C 180,E1 21208.03,E2 21208.03} C_VEL
LIN {X 0,Y 492.017,Z 443.215,A -85,B 0,C 180,E1 21205.565,E2 21205.565} C_VEL
LIN {X 0,Y 503.274,Z 461.442,A -85,B 0,C 180,E1 21203.254,E2 21203.254} C_VEL
LIN {X 0,Y 511.643,Z 476.212,A -85,B 0,C 180,E1 21201.651,E2 21201.651} C_VEL
LIN {X 0,Y 499.968,Z 722.479,A -85,B 0,C 180,E1 21197.87,E2 21197.87} C_VEL
LIN {X 0,Y 497.691,Z 766.294,A -85,B 0,C 180,E1 21197.164,E2 21197.164} C_VEL
LIN {X 0,Y 495.246,Z 790.201,A -85,B 0,C 180,E1 21196.621,E2 21196.621} C_VEL
LIN {X 0,Y 492.423,Z 811.739,A -85,B 0,C 180,E1 21195.986,E2 21195.986} C_VEL
LIN {X 0,Y 488.567,Z 835.485,A -85,B 0,C 180,E1 21195.082,E2 21195.082} C_VEL
LIN {X 0,Y 484.947,Z 854.788,A -85,B 0,C 180,E1 21194.179,E2 21194.179} C_VEL
LIN {X 0,Y 480.203,Z 877.436,A -85,B 0,C 180,E1 21192.913,E2 21192.913} C_VEL
LIN {X 0,Y 475.462,Z 897.422,A -85,B 0,C 180,E1 21191.567,E2 21191.567} C_VEL
LIN {X 0,Y 470.467,Z 917.266,A -85,B 0,C 180,E1 21190.009,E2 21190.009} C_VEL
LIN {X 0,Y 464.895,Z 937.64,A -85,B 0,C 180,E1 21188.117,E2 21188.117} C_VEL
LIN {X 0,Y 459.973,Z 955.021,A -85,B 0,C 180,E1 21186.246,E2 21186.246} C_VEL
LIN {X 0,Y 454.665,Z 973.247,A -85,B 0,C 180,E1 21183.958,E2 21183.958} C_VEL
LIN {X 0,Y 450.242,Z 988.386,A -85,B 0,C 180,E1 21181.758,E2 21181.758} C_VEL
LIN {X 0,Y 445.524,Z 1004.762,A -85,B 0,C 180,E1 21178.997,E2 21178.997} C_VEL
LIN {X 0,Y 441.972,Z 1017.607,A -85,B 0,C 180,E1 21176.467,E2 21176.467} C_VEL
LIN {X 0,Y 438.648,Z 1030.56,A -85,B 0,C 180,E1 21173.51,E2 21173.51} C_VEL
LIN {X 0,Y 436.221,Z 1041.033,A -85,B 0,C 180,E1 21170.67,E2 21170.67} C_VEL
LIN {X 0,Y 434.319,Z 1050.833,A -85,B 0,C 180,E1 21167.553,E2 21167.553} C_VEL
LIN {X 0,Y 433.067,Z 1058.69,A -85,B 0,C 180,E1 21164.439,E2 21164.439} C_VEL
LIN {X 0,Y 432.375,Z 1064.792,A -85,B 0,C 180,E1 21161.471,E2 21161.471} C_VEL
LIN {X 0,Y 432.028,Z 1069.722,A -85,B 0,C 180,E1 21158.25,E2 21158.25} C_VEL
LIN {X 0,Y 431.948,Z 1072.642,A -85,B 0,C 180,E1 21155.506,E2 21155.506} C_VEL
LIN {X 0,Y 431.942,Z 1074.478,A -85,B 0,C 180,E1 21152.654,E2 21152.654} C_VEL
LIN {X 0,Y 431.944,Z 1074.935,A -85,B 0,C 180,E1 21149.469,E2 21149.469} C_VEL
LIN {X 0,Y 431.947,Z 1074.097,A -85,B 0,C 180,E1 21146.815,E2 21146.815} C_VEL
LIN {X 0,Y 431.957,Z 1072.052,A -85,B 0,C 180,E1 21144.021,E2 21144.021} C_VEL
LIN {X 0,Y 432.098,Z 1067.939,A -85,B 0,C 180,E1 21140.678,E2 21140.678} C_VEL
LIN {X 0,Y 432.468,Z 1063.258,A -85,B 0,C 180,E1 21137.961,E2 21137.961} C_VEL
LIN {X 0,Y 433.263,Z 1056.581,A -85,B 0,C 180,E1 21134.884,E2 21134.884} C_VEL
LIN {X 0,Y 434.613,Z 1047.978,A -85,B 0,C 180,E1 21131.767,E2 21131.767} C_VEL
LIN {X 0,Y 436.447,Z 1038.639,A -85,B 0,C 180,E1 21128.919,E2 21128.919} C_VEL
LIN {X 0,Y 439.195,Z 1026.418,A -85,B 0,C 180,E1 21125.808,E2 21125.808} C_VEL
LIN {X 0,Y 442.123,Z 1014.703,A -85,B 0,C 180,E1 21123.253,E2 21123.253} C_VEL
LIN {X 0,Y 446.307,Z 998.982,A -85,B 0,C 180,E1 21120.322,E2 21120.322} C_VEL
LIN {X 0,Y 450.249,Z 984.69,A -85,B 0,C 180,E1 21118.031,E2 21118.031} C_VEL
LIN {X 0,Y 455.37,Z 966.303,A -85,B 0,C 180,E1 21115.493,E2 21115.493} C_VEL
LIN {X 0,Y 459.837,Z 950.082,A -85,B 0,C 180,E1 21113.567,E2 21113.567} C_VEL
LIN {X 0,Y 465.189,Z 930.126,A -85,B 0,C 180,E1 21111.519,E2 21111.519} C_VEL
LIN {X 0,Y 469.751,Z 912.077,A -85,B 0,C 180,E1 21109.937,E2 21109.937} C_VEL
LIN {X 0,Y 474.735,Z 891.264,A -85,B 0,C 180,E1 21108.355,E2 21108.355} C_VEL
LIN {X 0,Y 479.385,Z 869.689,A -85,B 0,C 180,E1 21106.996,E2 21106.996} C_VEL
LIN {X 0,Y 483.602,Z 848.094,A -85,B 0,C 180,E1 21105.845,E2 21105.845} C_VEL
LIN {X 0,Y 487.513,Z 824.79,A -85,B 0,C 180,E1 21104.84,E2 21104.84} C_VEL
LIN {X 0,Y 490.647,Z 802.953,A -85,B 0,C 180,E1 21104.086,E2 21104.086} C_VEL
LIN {X 0,Y 493.595,Z 776.73,A -85,B 0,C 180,E1 21103.403,E2 21103.403} C_VEL
LIN {X 0,Y 495.266,Z 754.369,A -85,B 0,C 180,E1 21102.977,E2 21102.977} C_VEL
LIN {X 0,Y 506.399,Z 505.651,A -85,B 0,C 180,E1 21099.158,E2 21099.158} C_VEL
LIN {X 0,Y 507.752,Z 473.861,A -85,B 0,C 180,E1 21098.654,E2 21098.654} C_VEL
LIN {X 0,Y 496.766,Z 454.506,A -85,B 0,C 180,E1 21096.659,E2 21096.659} C_VEL
LIN {X 0,Y 485.526,Z 436.238,A -85,B 0,C 180,E1 21094.459,E2 21094.459} C_VEL
LIN {X 0,Y 474.396,Z 419.479,A -85,B 0,C 180,E1 21092.083,E2 21092.083} C_VEL
LIN {X 0,Y 464.351,Z 405.315,A -85,B 0,C 180,E1 21089.723,E2 21089.723} C_VEL
LIN {X 0,Y 456.195,Z 394.492,A -85,B 0,C 180,E1 21087.618,E2 21087.618} C_VEL
LIN {X 0,Y 451.654,Z 388.602,A -85,B 0,C 180,E1 21086.352,E2 21086.352} C_VEL
LIN {X 0,Y 448.444,Z 384.751,A -85,B 0,C 180,E1 21085.418,E2 21085.418} C_VEL
LIN {X 0,Y 444.619,Z 379.774,A -85,B 0,C 180,E1 21084.231,E2 21084.231} C_VEL
LIN {X 0,Y 441.559,Z 377.023,A -85,B 0,C 180,E1 21083.275,E2 21083.275} C_VEL
LIN {X 0,Y 439.696,Z 373.645,A -85,B 0,C 180,E1 21082.601,E2 21082.601} C_VEL
LIN {X 0,Y 436.563,Z 371.7,A -85,B 0,C 180,E1 21081.568,E2 21081.568} C_VEL
LIN {X 0,Y 434.835,Z 368.902,A -85,B 0,C 180,E1 21080.898,E2 21080.898} C_VEL
LIN {X 0,Y 434.414,Z 367.107,A -85,B 0,C 180,E1 21080.655,E2 21080.655} C_VEL
LIN {X 0,Y 434.406,Z 367.12,A -85,B 0,C 180,E1 21076.759,E2 21076.759} C_VEL
LIN {X 0,Y 434.37,Z 367.098,A -85,B 0,C 180,E1 21073.165,E2 21073.165} C_VEL
LIN {X 0,Y 434.36,Z 367.086,A -85,B 0,C 180,E1 21069.407,E2 21069.407} C_VEL
LIN {X 0,Y 434.362,Z 367.096,A -85,B 0,C 180,E1 21065.548,E2 21065.548} C_VEL
LIN {X 0,Y 434.383,Z 367.125,A -85,B 0,C 180,E1 21061.847,E2 21061.847} C_VEL
LIN {X 0,Y 434.41,Z 367.084,A -85,B 0,C 180,E1 21058.285,E2 21058.285} C_VEL
LIN {X 0,Y 434.396,Z 367.082,A -85,B 0,C 180,E1 21054.452,E2 21054.452} C_VEL
LIN {X 0,Y 434.37,Z 367.117,A -85,B 0,C 180,E1 21050.861,E2 21050.861} C_VEL
LIN {X 0,Y 434.365,Z 367.108,A -85,B 0,C 180,E1 21047.098,E2 21047.098} C_VEL
LIN {X 0,Y 434.373,Z 367.087,A -85,B 0,C 180,E1 21043.415,E2 21043.415} C_VEL
LIN {X 0,Y 434.407,Z 367.088,A -85,B 0,C 180,E1 21039.802,E2 21039.802} C_VEL
LIN {X 0,Y 434.403,Z 367.369,A -85,B 0,C 180,E1 21036.893,E2 21036.893} C_VEL
LIN {X 0,Y 435.405,Z 370.151,A -85,B 0,C 180,E1 21036.448,E2 21036.448} C_VEL
LIN {X 0,Y 438.005,Z 372.837,A -85,B 0,C 180,E1 21035.522,E2 21035.522} C_VEL
LIN {X 0,Y 440.013,Z 374.076,A -85,B 0,C 180,E1 21034.871,E2 21034.871} C_VEL
LIN {X 0,Y 442.037,Z 377.566,A -85,B 0,C 180,E1 21034.151,E2 21034.151} C_VEL
LIN {X 0,Y 445.524,Z 380.607,A -85,B 0,C 180,E1 21033.077,E2 21033.077} C_VEL
LIN {X 0,Y 448.383,Z 384.646,A -85,B 0,C 180,E1 21032.184,E2 21032.184} C_VEL
LIN {X 0,Y 450.75,Z 386.798,A -85,B 0,C 180,E1 21031.515,E2 21031.515} C_VEL
LIN {X 0,Y 454.01,Z 391.044,A -85,B 0,C 180,E1 21030.585,E2 21030.585} C_VEL
LIN {X 0,Y 455.822,Z 392.993,A -85,B 0,C 180,E1 21030.099,E2 21030.099} C_VEL
LIN {X 0,Y 459.596,Z 397.562,A -85,B 0,C 180,E1 21029.107,E2 21029.107} C_VEL
LIN {X 0,Y 465.963,Z 405.657,A -85,B 0,C 180,E1 21027.52,E2 21027.52} C_VEL
LIN {X 0,Y 473.123,Z 414.677,A -85,B 0,C 180,E1 21025.868,E2 21025.868} C_VEL
LIN {X 0,Y 484.592,Z 430.179,A -85,B 0,C 180,E1 21023.43,E2 21023.43} C_VEL
LIN {X 0,Y 496.643,Z 447.502,A -85,B 0,C 180,E1 21021.105,E2 21021.105} C_VEL
LIN {X 0,Y 506.73,Z 463.438,A -85,B 0,C 180,E1 21019.296,E2 21019.296} C_VEL
LIN {X 0,Y 508.051,Z 466.028,A -85,B 0,C 180,E1 21019.058,E2 21019.058} C_VEL
LIN {X 0,Y 496.638,Z 718.586,A -85,B 0,C 180,E1 21015.192,E2 21015.192} C_VEL
LIN {X 0,Y 494.781,Z 751.494,A -85,B 0,C 180,E1 21014.633,E2 21014.633} C_VEL
LIN {X 0,Y 492.67,Z 773.612,A -85,B 0,C 180,E1 21014.101,E2 21014.101} C_VEL
LIN {X 0,Y 489.658,Z 798.079,A -85,B 0,C 180,E1 21013.323,E2 21013.323} C_VEL
LIN {X 0,Y 486.432,Z 818.959,A -85,B 0,C 180,E1 21012.474,E2 21012.474} C_VEL
LIN {X 0,Y 482.523,Z 841.197,A -85,B 0,C 180,E1 21011.379,E2 21011.379} C_VEL
LIN {X 0,Y 478.106,Z 862.578,A -85,B 0,C 180,E1 21010.101,E2 21010.101} C_VEL
LIN {X 0,Y 473.753,Z 881.913,A -85,B 0,C 180,E1 21008.74,E2 21008.74} C_VEL
LIN {X 0,Y 468.395,Z 903.636,A -85,B 0,C 180,E1 21006.936,E2 21006.936} C_VEL
LIN {X 0,Y 463.901,Z 920.654,A -85,B 0,C 180,E1 21005.285,E2 21005.285} C_VEL
LIN {X 0,Y 458.704,Z 939.537,A -85,B 0,C 180,E1 21003.17,E2 21003.17} C_VEL
LIN {X 0,Y 453.988,Z 955.906,A -85,B 0,C 180,E1 21001.022,E2 21001.022} C_VEL
LIN {X 0,Y 449.39,Z 972.081,A -85,B 0,C 180,E1 20998.579,E2 20998.579} C_VEL
LIN {X 0,Y 445.178,Z 986.714,A -85,B 0,C 180,E1 20995.975,E2 20995.975} C_VEL
LIN {X 0,Y 441.519,Z 1000.18,A -85,B 0,C 180,E1 20993.207,E2 20993.207} C_VEL
LIN {X 0,Y 438.535,Z 1011.589,A -85,B 0,C 180,E1 20990.417,E2 20990.417} C_VEL
LIN {X 0,Y 436.196,Z 1021.758,A -85,B 0,C 180,E1 20987.522,E2 20987.522} C_VEL
LIN {X 0,Y 434.361,Z 1030.763,A -85,B 0,C 180,E1 20984.395,E2 20984.395} C_VEL
LIN {X 0,Y 433.253,Z 1037.454,A -85,B 0,C 180,E1 20981.583,E2 20981.583} C_VEL
LIN {X 0,Y 432.461,Z 1043.675,A -85,B 0,C 180,E1 20978.242,E2 20978.242} C_VEL
LIN {X 0,Y 432.383,Z 1044.478,A -85,B 0,C 180,E1 20977.711,E2 20977.711} C_VEL
LIN {X 0,Y 431.252,Z 1046.049,A -85,B 0,C 180,E1 20976.712,E2 20976.712} C_VEL
LIN {X 0,Y 424.68,Z 1049.373,A -85,B 0,C 180,E1 20973.957,E2 20973.957} C_VEL
LIN {X 0,Y 424.015,Z 1050.046,A -85,B 0,C 180,E1 20973.139,E2 20973.139} C_VEL
LIN {X 0,Y 423.97,Z 1051.839,A -85,B 0,C 180,E1 20970,E2 20970} C_VEL
LIN {X 0,Y 423.952,Z 1052.046,A -85,B 0,C 180,E1 20966.89,E2 20966.89} C_VEL
LIN {X 0,Y 423.99,Z 1051.15,A -85,B 0,C 180,E1 20964.18,E2 20964.18} C_VEL
LIN {X 0,Y 424.116,Z 1048.864,A -85,B 0,C 180,E1 20961.048,E2 20961.048} C_VEL
LIN {X 0,Y 424.471,Z 1044.87,A -85,B 0,C 180,E1 20957.846,E2 20957.846} C_VEL
LIN {X 0,Y 425.153,Z 1039.888,A -85,B 0,C 180,E1 20954.867,E2 20954.867} C_VEL
LIN {X 0,Y 426.447,Z 1032.657,A -85,B 0,C 180,E1 20951.547,E2 20951.547} C_VEL
LIN {X 0,Y 428.084,Z 1025.127,A -85,B 0,C 180,E1 20948.743,E2 20948.743} C_VEL
LIN {X 0,Y 430.657,Z 1015.015,A -85,B 0,C 180,E1 20945.589,E2 20945.589} C_VEL
LIN {X 0,Y 433.776,Z 1003.834,A -85,B 0,C 180,E1 20942.696,E2 20942.696} C_VEL
LIN {X 0,Y 437.683,Z 990.946,A -85,B 0,C 180,E1 20939.828,E2 20939.828} C_VEL
LIN {X 0,Y 441.9,Z 977.282,A -85,B 0,C 180,E1 20937.263,E2 20937.263} C_VEL
LIN {X 0,Y 446.55,Z 962.651,A -85,B 0,C 180,E1 20934.868,E2 20934.868} C_VEL
LIN {X 0,Y 451.957,Z 945.292,A -85,B 0,C 180,E1 20932.446,E2 20932.446} C_VEL
LIN {X 0,Y 457.023,Z 928.778,A -85,B 0,C 180,E1 20930.457,E2 20930.457} C_VEL
LIN {X 0,Y 462.732,Z 909.231,A -85,B 0,C 180,E1 20928.442,E2 20928.442} C_VEL
LIN {X 0,Y 467.522,Z 891.777,A -85,B 0,C 180,E1 20926.897,E2 20926.897} C_VEL
LIN {X 0,Y 472.813,Z 871.108,A -85,B 0,C 180,E1 20925.319,E2 20925.319} C_VEL
LIN {X 0,Y 477.553,Z 850.328,A -85,B 0,C 180,E1 20923.996,E2 20923.996} C_VEL
LIN {X 0,Y 481.999,Z 828.767,A -85,B 0,C 180,E1 20922.834,E2 20922.834} C_VEL
LIN {X 0,Y 485.904,Z 806.181,A -85,B 0,C 180,E1 20921.848,E2 20921.848} C_VEL
LIN {X 0,Y 488.82,Z 786.379,A -85,B 0,C 180,E1 20921.143,E2 20921.143} C_VEL
LIN {X 0,Y 491.754,Z 761.454,A -85,B 0,C 180,E1 20920.452,E2 20920.452} C_VEL
LIN {X 0,Y 493.545,Z 739.017,A -85,B 0,C 180,E1 20920.002,E2 20920.002} C_VEL
LIN {X 0,Y 505.626,Z 494.827,A -85,B 0,C 180,E1 20916.221,E2 20916.221} C_VEL
LIN {X 0,Y 506.705,Z 471.513,A -85,B 0,C 180,E1 20915.844,E2 20915.844} C_VEL
LIN {X 0,Y 496.592,Z 455.764,A -85,B 0,C 180,E1 20913.865,E2 20913.865} C_VEL
LIN {X 0,Y 485.373,Z 439.786,A -85,B 0,C 180,E1 20911.482,E2 20911.482} C_VEL
LIN {X 0,Y 475.719,Z 426.782,A -85,B 0,C 180,E1 20909.22,E2 20909.22} C_VEL
LIN {X 0,Y 467.493,Z 416.348,A -85,B 0,C 180,E1 20907.102,E2 20907.102} C_VEL
LIN {X 0,Y 463.038,Z 410.841,A -85,B 0,C 180,E1 20905.862,E2 20905.862} C_VEL
LIN {X 0,Y 458.779,Z 405.565,A -85,B 0,C 180,E1 20904.6,E2 20904.6} C_VEL
LIN {X 0,Y 455.074,Z 401.044,A -85,B 0,C 180,E1 20903.434,E2 20903.434} C_VEL
LIN {X 0,Y 450.464,Z 395.877,A -85,B 0,C 180,E1 20901.895,E2 20901.895} C_VEL
LIN {X 0,Y 449.141,Z 394.029,A -85,B 0,C 180,E1 20901.414,E2 20901.414} C_VEL
LIN {X 0,Y 445.811,Z 390.841,A -85,B 0,C 180,E1 20900.206,E2 20900.206} C_VEL
LIN {X 0,Y 444.018,Z 387.983,A -85,B 0,C 180,E1 20899.468,E2 20899.468} C_VEL
LIN {X 0,Y 440.775,Z 385.427,A -85,B 0,C 180,E1 20898.175,E2 20898.175} C_VEL
LIN {X 0,Y 438.663,Z 381.728,A -85,B 0,C 180,E1 20897.169,E2 20897.169} C_VEL
LIN {X 0,Y 434.968,Z 379.222,A -85,B 0,C 180,E1 20895.466,E2 20895.466} C_VEL
LIN {X 0,Y 433.08,Z 376.196,A -85,B 0,C 180,E1 20894.405,E2 20894.405} C_VEL
LIN {X 0,Y 432.523,Z 374.865,A -85,B 0,C 180,E1 20894.048,E2 20894.048} C_VEL
LIN {X 0,Y 429.116,Z 373.125,A -85,B 0,C 180,E1 20892.105,E2 20892.105} C_VEL
LIN {X 0,Y 427.026,Z 370.28,A -85,B 0,C 180,E1 20890.592,E2 20890.592} C_VEL
LIN {X 0,Y 426.463,Z 368.08,A -85,B 0,C 180,E1 20889.992,E2 20889.992} C_VEL
LIN {X 0,Y 426.437,Z 368.086,A -85,B 0,C 180,E1 20886.327,E2 20886.327} C_VEL
LIN {X 0,Y 426.424,Z 368.095,A -85,B 0,C 180,E1 20882.553,E2 20882.553} C_VEL
LIN {X 0,Y 426.427,Z 368.106,A -85,B 0,C 180,E1 20878.791,E2 20878.791} C_VEL
LIN {X 0,Y 426.437,Z 368.114,A -85,B 0,C 180,E1 20875.023,E2 20875.023} C_VEL
LIN {X 0,Y 426.465,Z 368.095,A -85,B 0,C 180,E1 20871.37,E2 20871.37} C_VEL
LIN {X 0,Y 426.455,Z 368.313,A -85,B 0,C 180,E1 20868.298,E2 20868.298} C_VEL
LIN {X 0,Y 427.411,Z 370.977,A -85,B 0,C 180,E1 20867.434,E2 20867.434} C_VEL
LIN {X 0,Y 429.495,Z 373.449,A -85,B 0,C 180,E1 20865.988,E2 20865.988} C_VEL
LIN {X 0,Y 432.77,Z 375.179,A -85,B 0,C 180,E1 20864.145,E2 20864.145} C_VEL
LIN {X 0,Y 434.443,Z 378.617,A -85,B 0,C 180,E1 20863.142,E2 20863.142} C_VEL
LIN {X 0,Y 437.331,Z 381.042,A -85,B 0,C 180,E1 20861.746,E2 20861.746} C_VEL
LIN {X 0,Y 438.682,Z 381.886,A -85,B 0,C 180,E1 20861.15,E2 20861.15} C_VEL
LIN {X 0,Y 440.746,Z 385.354,A -85,B 0,C 180,E1 20860.174,E2 20860.174} C_VEL
LIN {X 0,Y 444.521,Z 388.609,A -85,B 0,C 180,E1 20858.664,E2 20858.664} C_VEL
LIN {X 0,Y 447.227,Z 392.486,A -85,B 0,C 180,E1 20857.592,E2 20857.592} C_VEL
LIN {X 0,Y 449.677,Z 394.898,A -85,B 0,C 180,E1 20856.719,E2 20856.719} C_VEL
LIN {X 0,Y 457.541,Z 404.981,A -85,B 0,C 180,E1 20854.083,E2 20854.083} C_VEL
LIN {X 0,Y 462.492,Z 411.613,A -85,B 0,C 180,E1 20852.581,E2 20852.581} C_VEL
LIN {X 0,Y 468.947,Z 420.397,A -85,B 0,C 180,E1 20850.773,E2 20850.773} C_VEL
LIN {X 0,Y 478.305,Z 433.707,A -85,B 0,C 180,E1 20848.386,E2 20848.386} C_VEL
LIN {X 0,Y 488.863,Z 449.818,A -85,B 0,C 180,E1 20845.95,E2 20845.95} C_VEL
LIN {X 0,Y 499.986,Z 468.064,A -85,B 0,C 180,E1 20843.615,E2 20843.615} C_VEL
LIN {X 0,Y 506.594,Z 479.918,A -85,B 0,C 180,E1 20842.312,E2 20842.312} C_VEL
LIN {X 0,Y 494.495,Z 726.812,A -85,B 0,C 180,E1 20838.499,E2 20838.499} C_VEL
LIN {X 0,Y 492.31,Z 766.561,A -85,B 0,C 180,E1 20837.85,E2 20837.85} C_VEL
LIN {X 0,Y 489.836,Z 790.096,A -85,B 0,C 180,E1 20837.312,E2 20837.312} C_VEL
LIN {X 0,Y 486.878,Z 812.003,A -85,B 0,C 180,E1 20836.663,E2 20836.663} C_VEL
LIN {X 0,Y 482.863,Z 835.876,A -85,B 0,C 180,E1 20835.745,E2 20835.745} C_VEL
LIN {X 0,Y 479.188,Z 854.851,A -85,B 0,C 180,E1 20834.852,E2 20834.852} C_VEL
LIN {X 0,Y 474.298,Z 877.442,A -85,B 0,C 180,E1 20833.58,E2 20833.58} C_VEL
LIN {X 0,Y 469.42,Z 897.339,A -85,B 0,C 180,E1 20832.231,E2 20832.231} C_VEL
LIN {X 0,Y 464.24,Z 917.229,A -85,B 0,C 180,E1 20830.657,E2 20830.657} C_VEL
LIN {X 0,Y 458.654,Z 936.961,A -85,B 0,C 180,E1 20828.812,E2 20828.812} C_VEL
LIN {X 0,Y 453.696,Z 953.814,A -85,B 0,C 180,E1 20826.989,E2 20826.989} C_VEL
LIN {X 0,Y 447.752,Z 973.418,A -85,B 0,C 180,E1 20824.51,E2 20824.51} C_VEL
LIN {X 0,Y 443.226,Z 988.268,A -85,B 0,C 180,E1 20822.321,E2 20822.321} C_VEL
LIN {X 0,Y 438.297,Z 1004.625,A -85,B 0,C 180,E1 20819.522,E2 20819.522} C_VEL
LIN {X 0,Y 434.57,Z 1017.461,A -85,B 0,C 180,E1 20816.954,E2 20816.954} C_VEL
LIN {X 0,Y 431.071,Z 1030.399,A -85,B 0,C 180,E1 20813.949,E2 20813.949} C_VEL
LIN {X 0,Y 428.483,Z 1040.986,A -85,B 0,C 180,E1 20811.024,E2 20811.024} C_VEL
LIN {X 0,Y 426.465,Z 1050.772,A -85,B 0,C 180,E1 20807.84,E2 20807.84} C_VEL
LIN {X 0,Y 425.154,Z 1058.506,A -85,B 0,C 180,E1 20804.714,E2 20804.714} C_VEL
LIN {X 0,Y 424.411,Z 1064.603,A -85,B 0,C 180,E1 20801.69,E2 20801.69} C_VEL
LIN {X 0,Y 424.042,Z 1069.524,A -85,B 0,C 180,E1 20798.407,E2 20798.407} C_VEL
LIN {X 0,Y 423.95,Z 1072.375,A -85,B 0,C 180,E1 20795.685,E2 20795.685} C_VEL
LIN {X 0,Y 423.945,Z 1074.203,A -85,B 0,C 180,E1 20792.839,E2 20792.839} C_VEL
LIN {X 0,Y 423.947,Z 1074.742,A -85,B 0,C 180,E1 20789.595,E2 20789.595} C_VEL
LIN {X 0,Y 423.949,Z 1073.945,A -85,B 0,C 180,E1 20786.89,E2 20786.89} C_VEL
LIN {X 0,Y 423.955,Z 1072.058,A -85,B 0,C 180,E1 20784.179,E2 20784.179} C_VEL
LIN {X 0,Y 424.076,Z 1068.332,A -85,B 0,C 180,E1 20780.911,E2 20780.911} C_VEL
LIN {X 0,Y 424.478,Z 1063.328,A -85,B 0,C 180,E1 20777.898,E2 20777.898} C_VEL
LIN {X 0,Y 425.217,Z 1057.258,A -85,B 0,C 180,E1 20775.009,E2 20775.009} C_VEL
LIN {X 0,Y 426.677,Z 1048.368,A -85,B 0,C 180,E1 20771.64,E2 20771.64} C_VEL
LIN {X 0,Y 428.526,Z 1039.3,A -85,B 0,C 180,E1 20768.798,E2 20768.798} C_VEL
LIN {X 0,Y 431.5,Z 1026.713,A -85,B 0,C 180,E1 20765.494,E2 20765.494} C_VEL
LIN {X 0,Y 434.54,Z 1015.052,A -85,B 0,C 180,E1 20762.896,E2 20762.896} C_VEL
LIN {X 0,Y 438.889,Z 999.45,A -85,B 0,C 180,E1 20759.92,E2 20759.92} C_VEL
LIN {X 0,Y 443.114,Z 984.724,A -85,B 0,C 180,E1 20757.517,E2 20757.517} C_VEL
LIN {X 0,Y 448.571,Z 965.947,A -85,B 0,C 180,E1 20754.892,E2 20754.892} C_VEL
LIN {X 0,Y 453.173,Z 949.861,A -85,B 0,C 180,E1 20752.961,E2 20752.961} C_VEL
LIN {X 0,Y 458.698,Z 929.968,A -85,B 0,C 180,E1 20750.898,E2 20750.898} C_VEL
LIN {X 0,Y 463.716,Z 910.755,A -85,B 0,C 180,E1 20749.206,E2 20749.206} C_VEL
LIN {X 0,Y 468.837,Z 889.947,A -85,B 0,C 180,E1 20747.629,E2 20747.629} C_VEL
LIN {X 0,Y 473.443,Z 869.222,A -85,B 0,C 180,E1 20746.322,E2 20746.322} C_VEL
LIN {X 0,Y 477.832,Z 847.403,A -85,B 0,C 180,E1 20745.155,E2 20745.155} C_VEL
LIN {X 0,Y 481.835,Z 824.131,A -85,B 0,C 180,E1 20744.152,E2 20744.152} C_VEL
LIN {X 0,Y 485.048,Z 802.306,A -85,B 0,C 180,E1 20743.399,E2 20743.399} C_VEL
LIN {X 0,Y 488.038,Z 776.326,A -85,B 0,C 180,E1 20742.724,E2 20742.724} C_VEL
LIN {X 0,Y 489.749,Z 753.945,A -85,B 0,C 180,E1 20742.296,E2 20742.296} C_VEL
LIN {X 0,Y 501.263,Z 505.468,A -85,B 0,C 180,E1 20738.455,E2 20738.455} C_VEL
LIN {X 0,Y 502.5,Z 477.419,A -85,B 0,C 180,E1 20738.007,E2 20738.007} C_VEL
LIN {X 0,Y 491.324,Z 457.681,A -85,B 0,C 180,E1 20735.907,E2 20735.907} C_VEL
LIN {X 0,Y 480.153,Z 439.521,A -85,B 0,C 180,E1 20733.637,E2 20733.637} C_VEL
LIN {X 0,Y 468.819,Z 422.405,A -85,B 0,C 180,E1 20731.109,E2 20731.109} C_VEL
LIN {X 0,Y 458.193,Z 407.553,A -85,B 0,C 180,E1 20728.478,E2 20728.478} C_VEL
LIN {X 0,Y 449.566,Z 396.077,A -85,B 0,C 180,E1 20726.093,E2 20726.093} C_VEL
LIN {X 0,Y 445.699,Z 391.494,A -85,B 0,C 180,E1 20724.946,E2 20724.946} C_VEL
LIN {X 0,Y 442.505,Z 387.216,A -85,B 0,C 180,E1 20723.929,E2 20723.929} C_VEL
LIN {X 0,Y 439.228,Z 384.03,A -85,B 0,C 180,E1 20722.874,E2 20722.874} C_VEL
LIN {X 0,Y 437.634,Z 381.227,A -85,B 0,C 180,E1 20722.289,E2 20722.289} C_VEL
LIN {X 0,Y 434.401,Z 378.872,A -85,B 0,C 180,E1 20721.185,E2 20721.185} C_VEL
LIN {X 0,Y 432.444,Z 375.567,A -85,B 0,C 180,E1 20720.399,E2 20720.399} C_VEL
LIN {X 0,Y 432.079,Z 374.761,A -85,B 0,C 180,E1 20720.241,E2 20720.241} C_VEL
LIN {X 0,Y 428.916,Z 372.928,A -85,B 0,C 180,E1 20719.049,E2 20719.049} C_VEL
LIN {X 0,Y 426.898,Z 369.924,A -85,B 0,C 180,E1 20718.151,E2 20718.151} C_VEL
LIN {X 0,Y 426.426,Z 368.087,A -85,B 0,C 180,E1 20717.826,E2 20717.826} C_VEL
LIN {X 0,Y 426.442,Z 368.074,A -85,B 0,C 180,E1 20714.114,E2 20714.114} C_VEL
LIN {X 0,Y 426.464,Z 368.076,A -85,B 0,C 180,E1 20710.401,E2 20710.401} C_VEL
LIN {X 0,Y 426.47,Z 368.105,A -85,B 0,C 180,E1 20706.597,E2 20706.597} C_VEL
LIN {X 0,Y 426.446,Z 368.091,A -85,B 0,C 180,E1 20702.756,E2 20702.756} C_VEL
LIN {X 0,Y 426.423,Z 368.071,A -85,B 0,C 180,E1 20699.059,E2 20699.059} C_VEL
LIN {X 0,Y 426.423,Z 368.086,A -85,B 0,C 180,E1 20695.24,E2 20695.24} C_VEL
LIN {X 0,Y 426.434,Z 368.114,A -85,B 0,C 180,E1 20691.505,E2 20691.505} C_VEL
LIN {X 0,Y 426.454,Z 368.076,A -85,B 0,C 180,E1 20687.818,E2 20687.818} C_VEL
LIN {X 0,Y 426.473,Z 368.07,A -85,B 0,C 180,E1 20684.079,E2 20684.079} C_VEL
LIN {X 0,Y 426.458,Z 368.084,A -85,B 0,C 180,E1 20680.267,E2 20680.267} C_VEL
LIN {X 0,Y 426.48,Z 368.249,A -85,B 0,C 180,E1 20679.678,E2 20679.678} C_VEL
LIN {X 0,Y 427.365,Z 370.958,A -85,B 0,C 180,E1 20679.204,E2 20679.204} C_VEL
LIN {X 0,Y 429.721,Z 373.581,A -85,B 0,C 180,E1 20678.215,E2 20678.215} C_VEL
LIN {X 0,Y 432.238,Z 375.085,A -85,B 0,C 180,E1 20677.274,E2 20677.274} C_VEL
LIN {X 0,Y 434.091,Z 378.452,A -85,B 0,C 180,E1 20676.516,E2 20676.516} C_VEL
LIN {X 0,Y 437.283,Z 381.067,A -85,B 0,C 180,E1 20675.407,E2 20675.407} C_VEL
LIN {X 0,Y 437.991,Z 381.856,A -85,B 0,C 180,E1 20675.162,E2 20675.162} C_VEL
LIN {X 0,Y 440.624,Z 385.652,A -85,B 0,C 180,E1 20674.242,E2 20674.242} C_VEL
LIN {X 0,Y 443.311,Z 388.033,A -85,B 0,C 180,E1 20673.402,E2 20673.402} C_VEL
LIN {X 0,Y 446.548,Z 392.308,A -85,B 0,C 180,E1 20672.386,E2 20672.386} C_VEL
LIN {X 0,Y 448.568,Z 394.354,A -85,B 0,C 180,E1 20671.799,E2 20671.799} C_VEL
LIN {X 0,Y 452.237,Z 398.813,A -85,B 0,C 180,E1 20670.749,E2 20670.749} C_VEL
LIN {X 0,Y 458.514,Z 406.657,A -85,B 0,C 180,E1 20669.062,E2 20669.062} C_VEL
LIN {X 0,Y 463.411,Z 412.851,A -85,B 0,C 180,E1 20667.832,E2 20667.832} C_VEL
LIN {X 0,Y 470.492,Z 421.952,A -85,B 0,C 180,E1 20666.165,E2 20666.165} C_VEL
LIN {X 0,Y 481.23,Z 436.582,A -85,B 0,C 180,E1 20663.836,E2 20663.836} C_VEL
LIN {X 0,Y 493.209,Z 454.026,A -85,B 0,C 180,E1 20661.472,E2 20661.472} C_VEL
LIN {X 0,Y 502.801,Z 469.369,A -85,B 0,C 180,E1 20659.713,E2 20659.713} C_VEL
LIN {X 0,Y 491.235,Z 716.868,A -85,B 0,C 180,E1 20655.897,E2 20655.897} C_VEL
LIN {X 0,Y 489.314,Z 750.771,A -85,B 0,C 180,E1 20655.326,E2 20655.326} C_VEL
LIN {X 0,Y 487.1,Z 773.465,A -85,B 0,C 180,E1 20654.781,E2 20654.781} C_VEL
LIN {X 0,Y 484.136,Z 797.158,A -85,B 0,C 180,E1 20654.033,E2 20654.033} C_VEL
LIN {X 0,Y 480.571,Z 819.588,A -85,B 0,C 180,E1 20653.117,E2 20653.117} C_VEL
LIN {X 0,Y 476.548,Z 841.777,A -85,B 0,C 180,E1 20652.015,E2 20652.015} C_VEL
LIN {X 0,Y 471.793,Z 863.976,A -85,B 0,C 180,E1 20650.67,E2 20650.67} C_VEL
LIN {X 0,Y 467.112,Z 884.074,A -85,B 0,C 180,E1 20649.23,E2 20649.23} C_VEL
LIN {X 0,Y 461.787,Z 904.731,A -85,B 0,C 180,E1 20647.477,E2 20647.477} C_VEL
LIN {X 0,Y 457.153,Z 921.671,A -85,B 0,C 180,E1 20645.808,E2 20645.808} C_VEL
LIN {X 0,Y 451.475,Z 941.415,A -85,B 0,C 180,E1 20643.544,E2 20643.544} C_VEL
LIN {X 0,Y 447.009,Z 956.39,A -85,B 0,C 180,E1 20641.543,E2 20641.543} C_VEL
LIN {X 0,Y 442.252,Z 972.428,A -85,B 0,C 180,E1 20639.084,E2 20639.084} C_VEL
LIN {X 0,Y 437.937,Z 986.804,A -85,B 0,C 180,E1 20636.49,E2 20636.49} C_VEL
LIN {X 0,Y 434.034,Z 1000.496,A -85,B 0,C 180,E1 20633.631,E2 20633.631} C_VEL
LIN {X 0,Y 430.845,Z 1012.145,A -85,B 0,C 180,E1 20630.727,E2 20630.727} C_VEL
LIN {X 0,Y 428.321,Z 1022.647,A -85,B 0,C 180,E1 20627.667,E2 20627.667} C_VEL
LIN {X 0,Y 426.445,Z 1031.387,A -85,B 0,C 180,E1 20624.53,E2 20624.53} C_VEL
LIN {X 0,Y 425.213,Z 1038.613,A -85,B 0,C 180,E1 20621.392,E2 20621.392} C_VEL
LIN {X 0,Y 424.455,Z 1044.329,A -85,B 0,C 180,E1 20618.125,E2 20618.125} C_VEL
LIN {X 0,Y 424.131,Z 1048.056,A -85,B 0,C 180,E1 20615.275,E2 20615.275} C_VEL
LIN {X 0,Y 424.015,Z 1050.046,A -85,B 0,C 180,E1 20613.139,E2 20613.139} C_VEL
LIN {X 0,Y 422.997,Z 1050.856,A -85,B 0,C 180,E1 20612.104,E2 20612.104} C_VEL
LIN {X 0,Y 416.589,Z 1052.175,A -85,B 0,C 180,E1 20609.255,E2 20609.255} C_VEL
LIN {X 0,Y 415.945,Z 1052.314,A -85,B 0,C 180,E1 20608.413,E2 20608.413} C_VEL
LIN {X 0,Y 415.972,Z 1051.818,A -85,B 0,C 180,E1 20605.036,E2 20605.036} C_VEL
LIN {X 0,Y 416.052,Z 1050.071,A -85,B 0,C 180,E1 20602.126,E2 20602.126} C_VEL
LIN {X 0,Y 416.291,Z 1047.175,A -85,B 0,C 180,E1 20599.202,E2 20599.202} C_VEL
LIN {X 0,Y 416.939,Z 1042.004,A -85,B 0,C 180,E1 20595.665,E2 20595.665} C_VEL
LIN {X 0,Y 417.92,Z 1036.341,A -85,B 0,C 180,E1 20592.742,E2 20592.742} C_VEL
LIN {X 0,Y 419.71,Z 1028.169,A -85,B 0,C 180,E1 20589.354,E2 20589.354} C_VEL
LIN {X 0,Y 421.935,Z 1019.336,A -85,B 0,C 180,E1 20586.391,E2 20586.391} C_VEL
LIN {X 0,Y 425.07,Z 1008.503,A -85,B 0,C 180,E1 20583.302,E2 20583.302} C_VEL
LIN {X 0,Y 428.861,Z 996.143,A -85,B 0,C 180,E1 20580.378,E2 20580.378} C_VEL
LIN {X 0,Y 433.239,Z 982.686,A -85,B 0,C 180,E1 20577.626,E2 20577.626} C_VEL
LIN {X 0,Y 438.22,Z 967.455,A -85,B 0,C 180,E1 20574.999,E2 20574.999} C_VEL
LIN {X 0,Y 443.075,Z 952.695,A -85,B 0,C 180,E1 20572.786,E2 20572.786} C_VEL
LIN {X 0,Y 449.039,Z 934.034,A -85,B 0,C 180,E1 20570.395,E2 20570.395} C_VEL
LIN {X 0,Y 454.325,Z 916.902,A -85,B 0,C 180,E1 20568.513,E2 20568.513} C_VEL
LIN {X 0,Y 460.35,Z 896.166,A -85,B 0,C 180,E1 20566.572,E2 20566.572} C_VEL
LIN {X 0,Y 465.245,Z 877.922,A -85,B 0,C 180,E1 20565.116,E2 20565.116} C_VEL
LIN {X 0,Y 470.527,Z 856.532,A -85,B 0,C 180,E1 20563.658,E2 20563.658} C_VEL
LIN {X 0,Y 475.1,Z 835.421,A -85,B 0,C 180,E1 20562.468,E2 20562.468} C_VEL
LIN {X 0,Y 479.346,Z 813.232,A -85,B 0,C 180,E1 20561.418,E2 20561.418} C_VEL
LIN {X 0,Y 482.959,Z 790.065,A -85,B 0,C 180,E1 20560.552,E2 20560.552} C_VEL
LIN {X 0,Y 485.748,Z 768.223,A -85,B 0,C 180,E1 20559.906,E2 20559.906} C_VEL
LIN {X 0,Y 488.106,Z 742.445,A -85,B 0,C 180,E1 20559.351,E2 20559.351} C_VEL
LIN {X 0,Y 500.072,Z 508.874,A -85,B 0,C 180,E1 20555.706,E2 20555.706} C_VEL
LIN {X 0,Y 501.723,Z 475.289,A -85,B 0,C 180,E1 20555.167,E2 20555.167} C_VEL
LIN {X 0,Y 491.043,Z 458.951,A -85,B 0,C 180,E1 20553.004,E2 20553.004} C_VEL
LIN {X 0,Y 480.225,Z 443.43,A -85,B 0,C 180,E1 20550.603,E2 20550.603} C_VEL
LIN {X 0,Y 469.661,Z 429.257,A -85,B 0,C 180,E1 20547.998,E2 20547.998} C_VEL
LIN {X 0,Y 460.98,Z 418.3,A -85,B 0,C 180,E1 20545.606,E2 20545.606} C_VEL
LIN {X 0,Y 456.288,Z 412.56,A -85,B 0,C 180,E1 20544.191,E2 20544.191} C_VEL
LIN {X 0,Y 451.936,Z 407.223,A -85,B 0,C 180,E1 20542.779,E2 20542.779} C_VEL
LIN {X 0,Y 448.305,Z 403.012,A -85,B 0,C 180,E1 20541.525,E2 20541.525} C_VEL
LIN {X 0,Y 447.158,Z 401.478,A -85,B 0,C 180,E1 20541.101,E2 20541.101} C_VEL
LIN {X 0,Y 443.662,Z 397.874,A -85,B 0,C 180,E1 20539.793,E2 20539.793} C_VEL
LIN {X 0,Y 442.109,Z 395.52,A -85,B 0,C 180,E1 20539.144,E2 20539.144} C_VEL
LIN {X 0,Y 438.805,Z 392.613,A -85,B 0,C 180,E1 20537.779,E2 20537.779} C_VEL
LIN {X 0,Y 436.709,Z 389.232,A -85,B 0,C 180,E1 20536.768,E2 20536.768} C_VEL
LIN {X 0,Y 433.255,Z 386.635,A -85,B 0,C 180,E1 20535.117,E2 20535.117} C_VEL
LIN {X 0,Y 431.273,Z 383.204,A -85,B 0,C 180,E1 20533.953,E2 20533.953} C_VEL
LIN {X 0,Y 430.836,Z 382.617,A -85,B 0,C 180,E1 20533.693,E2 20533.693} C_VEL
LIN {X 0,Y 427.55,Z 380.636,A -85,B 0,C 180,E1 20531.74,E2 20531.74} C_VEL
LIN {X 0,Y 425.626,Z 377.822,A -85,B 0,C 180,E1 20530.285,E2 20530.285} C_VEL
LIN {X 0,Y 424.917,Z 375.931,A -85,B 0,C 180,E1 20529.618,E2 20529.618} C_VEL
LIN {X 0,Y 420.979,Z 373.898,A -85,B 0,C 180,E1 20525.862,E2 20525.862} C_VEL
LIN {X 0,Y 418.688,Z 370.127,A -85,B 0,C 180,E1 20520.547,E2 20520.547} C_VEL
LIN {X 0,Y 418.612,Z 369.749,A -85,B 0,C 180,E1 20519.179,E2 20519.179} C_VEL
LIN {X 0,Y 418.818,Z 370.545,A -85,B 0,C 180,E1 20516.989,E2 20516.989} C_VEL
LIN {X 0,Y 423.403,Z 375.494,A -85,B 0,C 180,E1 20509.936,E2 20509.936} C_VEL
LIN {X 0,Y 425.089,Z 376.181,A -85,B 0,C 180,E1 20508.57,E2 20508.57} C_VEL
LIN {X 0,Y 426.592,Z 379.531,A -85,B 0,C 180,E1 20507.272,E2 20507.272} C_VEL
LIN {X 0,Y 429.411,Z 381.997,A -85,B 0,C 180,E1 20505.435,E2 20505.435} C_VEL
LIN {X 0,Y 431.26,Z 383.048,A -85,B 0,C 180,E1 20504.398,E2 20504.398} C_VEL
LIN {X 0,Y 433.226,Z 386.626,A -85,B 0,C 180,E1 20503.232,E2 20503.232} C_VEL
LIN {X 0,Y 436.396,Z 389.06,A -85,B 0,C 180,E1 20501.705,E2 20501.705} C_VEL
LIN {X 0,Y 437.075,Z 389.746,A -85,B 0,C 180,E1 20501.389,E2 20501.389} C_VEL
LIN {X 0,Y 439.638,Z 393.534,A -85,B 0,C 180,E1 20500.191,E2 20500.191} C_VEL
LIN {X 0,Y 442.695,Z 396.176,A -85,B 0,C 180,E1 20498.953,E2 20498.953} C_VEL
LIN {X 0,Y 445.617,Z 400.199,A -85,B 0,C 180,E1 20497.785,E2 20497.785} C_VEL
LIN {X 0,Y 448.034,Z 402.698,A -85,B 0,C 180,E1 20496.907,E2 20496.907} C_VEL
LIN {X 0,Y 455.36,Z 412.285,A -85,B 0,C 180,E1 20494.404,E2 20494.404} C_VEL
LIN {X 0,Y 460.534,Z 419.318,A -85,B 0,C 180,E1 20492.804,E2 20492.804} C_VEL
LIN {X 0,Y 466.618,Z 427.734,A -85,B 0,C 180,E1 20491.069,E2 20491.069} C_VEL
LIN {X 0,Y 475.649,Z 440.785,A -85,B 0,C 180,E1 20488.719,E2 20488.719} C_VEL
LIN {X 0,Y 485.731,Z 456.417,A -85,B 0,C 180,E1 20486.34,E2 20486.34} C_VEL
LIN {X 0,Y 496.408,Z 474.181,A -85,B 0,C 180,E1 20484.044,E2 20484.044} C_VEL
LIN {X 0,Y 501.607,Z 483.771,A -85,B 0,C 180,E1 20482.984,E2 20482.984} C_VEL
LIN {X 0,Y 489.101,Z 730.776,A -85,B 0,C 180,E1 20479.148,E2 20479.148} C_VEL
LIN {X 0,Y 486.969,Z 767.159,A -85,B 0,C 180,E1 20478.543,E2 20478.543} C_VEL
LIN {X 0,Y 484.48,Z 790.135,A -85,B 0,C 180,E1 20478.015,E2 20478.015} C_VEL
LIN {X 0,Y 481.317,Z 812.88,A -85,B 0,C 180,E1 20477.336,E2 20477.336} C_VEL
LIN {X 0,Y 477.335,Z 835.692,A -85,B 0,C 180,E1 20476.45,E2 20476.45} C_VEL
LIN {X 0,Y 473.495,Z 854.917,A -85,B 0,C 180,E1 20475.542,E2 20475.542} C_VEL
LIN {X 0,Y 468.282,Z 878.153,A -85,B 0,C 180,E1 20474.218,E2 20474.218} C_VEL
LIN {X 0,Y 463.407,Z 897.39,A -85,B 0,C 180,E1 20472.902,E2 20472.902} C_VEL
LIN {X 0,Y 457.88,Z 917.929,A -85,B 0,C 180,E1 20471.261,E2 20471.261} C_VEL
LIN {X 0,Y 451.979,Z 937.935,A -85,B 0,C 180,E1 20469.355,E2 20469.355} C_VEL
LIN {X 0,Y 446.652,Z 955.402,A -85,B 0,C 180,E1 20467.43,E2 20467.43} C_VEL
LIN {X 0,Y 441.063,Z 973.032,A -85,B 0,C 180,E1 20465.157,E2 20465.157} C_VEL
LIN {X 0,Y 436.255,Z 988.151,A -85,B 0,C 180,E1 20462.902,E2 20462.902} C_VEL
LIN {X 0,Y 431.109,Z 1004.489,A -85,B 0,C 180,E1 20460.065,E2 20460.065} C_VEL
LIN {X 0,Y 427.269,Z 1017.077,A -85,B 0,C 180,E1 20457.509,E2 20457.509} C_VEL
LIN {X 0,Y 423.524,Z 1030.24,A -85,B 0,C 180,E1 20454.403,E2 20454.403} C_VEL
LIN {X 0,Y 420.817,Z 1040.699,A -85,B 0,C 180,E1 20451.464,E2 20451.464} C_VEL
LIN {X 0,Y 418.67,Z 1050.475,A -85,B 0,C 180,E1 20448.232,E2 20448.232} C_VEL
LIN {X 0,Y 417.246,Z 1058.322,A -85,B 0,C 180,E1 20445,E2 20445} C_VEL
LIN {X 0,Y 416.452,Z 1064.415,A -85,B 0,C 180,E1 20441.916,E2 20441.916} C_VEL
LIN {X 0,Y 416.053,Z 1069.326,A -85,B 0,C 180,E1 20438.569,E2 20438.569} C_VEL
LIN {X 0,Y 415.953,Z 1072.173,A -85,B 0,C 180,E1 20435.795,E2 20435.795} C_VEL
LIN {X 0,Y 415.947,Z 1073.996,A -85,B 0,C 180,E1 20432.894,E2 20432.894} C_VEL
LIN {X 0,Y 415.951,Z 1074.526,A -85,B 0,C 180,E1 20429.587,E2 20429.587} C_VEL
LIN {X 0,Y 415.951,Z 1073.724,A -85,B 0,C 180,E1 20426.831,E2 20426.831} C_VEL
LIN {X 0,Y 415.958,Z 1071.831,A -85,B 0,C 180,E1 20424.067,E2 20424.067} C_VEL
LIN {X 0,Y 416.09,Z 1068.093,A -85,B 0,C 180,E1 20420.735,E2 20420.735} C_VEL
LIN {X 0,Y 416.522,Z 1063.082,A -85,B 0,C 180,E1 20417.664,E2 20417.664} C_VEL
LIN {X 0,Y 417.312,Z 1057.005,A -85,B 0,C 180,E1 20414.718,E2 20414.718} C_VEL
LIN {X 0,Y 418.828,Z 1048.271,A -85,B 0,C 180,E1 20411.343,E2 20411.343} C_VEL
LIN {X 0,Y 420.717,Z 1039.492,A -85,B 0,C 180,E1 20408.531,E2 20408.531} C_VEL
LIN {X 0,Y 423.668,Z 1027.59,A -85,B 0,C 180,E1 20405.308,E2 20405.308} C_VEL
LIN {X 0,Y 426.974,Z 1015.4,A -85,B 0,C 180,E1 20402.527,E2 20402.527} C_VEL
LIN {X 0,Y 431.27,Z 1000.7,A -85,B 0,C 180,E1 20399.64,E2 20399.64} C_VEL
LIN {X 0,Y 435.756,Z 985.622,A -85,B 0,C 180,E1 20397.122,E2 20397.122} C_VEL
LIN {X 0,Y 440.916,Z 968.695,A -85,B 0,C 180,E1 20394.671,E2 20394.671} C_VEL
LIN {X 0,Y 446.124,Z 951.105,A -85,B 0,C 180,E1 20392.506,E2 20392.506} C_VEL
LIN {X 0,Y 451.673,Z 932.049,A -85,B 0,C 180,E1 20390.472,E2 20390.472} C_VEL
LIN {X 0,Y 457.131,Z 911.839,A -85,B 0,C 180,E1 20388.657,E2 20388.657} C_VEL
LIN {X 0,Y 462.399,Z 891.244,A -85,B 0,C 180,E1 20387.066,E2 20387.066} C_VEL
LIN {X 0,Y 467.35,Z 869.768,A -85,B 0,C 180,E1 20385.69,E2 20385.69} C_VEL
LIN {X 0,Y 471.676,Z 848.949,A -85,B 0,C 180,E1 20384.562,E2 20384.562} C_VEL
LIN {X 0,Y 476.012,Z 824.836,A -85,B 0,C 180,E1 20383.501,E2 20383.501} C_VEL
LIN {X 0,Y 479.336,Z 802.967,A -85,B 0,C 180,E1 20382.738,E2 20382.738} C_VEL
LIN {X 0,Y 482.499,Z 776.475,A -85,B 0,C 180,E1 20382.041,E2 20382.041} C_VEL
LIN {X 0,Y 484.261,Z 754.165,A -85,B 0,C 180,E1 20381.611,E2 20381.611} C_VEL
LIN {X 0,Y 496.168,Z 506.014,A -85,B 0,C 180,E1 20377.749,E2 20377.749} C_VEL
LIN {X 0,Y 497.264,Z 480.875,A -85,B 0,C 180,E1 20377.337,E2 20377.337} C_VEL
LIN {X 0,Y 485.976,Z 460.861,A -85,B 0,C 180,E1 20375.141,E2 20375.141} C_VEL
LIN {X 0,Y 475.949,Z 444.657,A -85,B 0,C 180,E1 20373.036,E2 20373.036} C_VEL
LIN {X 0,Y 465.74,Z 428.971,A -85,B 0,C 180,E1 20370.692,E2 20370.692} C_VEL
LIN {X 0,Y 455.376,Z 414.304,A -85,B 0,C 180,E1 20368.063,E2 20368.063} C_VEL
LIN {X 0,Y 446.885,Z 402.869,A -85,B 0,C 180,E1 20365.655,E2 20365.655} C_VEL
LIN {X 0,Y 440.971,Z 395.228,A -85,B 0,C 180,E1 20363.804,E2 20363.804} C_VEL
LIN {X 0,Y 436.919,Z 391.036,A -85,B 0,C 180,E1 20362.469,E2 20362.469} C_VEL
LIN {X 0,Y 435.592,Z 388.754,A -85,B 0,C 180,E1 20361.973,E2 20361.973} C_VEL
LIN {X 0,Y 432.26,Z 386.031,A -85,B 0,C 180,E1 20360.798,E2 20360.798} C_VEL
LIN {X 0,Y 429.94,Z 382.324,A -85,B 0,C 180,E1 20359.849,E2 20359.849} C_VEL
LIN {X 0,Y 426.729,Z 379.982,A -85,B 0,C 180,E1 20358.583,E2 20358.583} C_VEL
LIN {X 0,Y 424.725,Z 376.641,A -85,B 0,C 180,E1 20357.644,E2 20357.644} C_VEL
LIN {X 0,Y 424.263,Z 375.798,A -85,B 0,C 180,E1 20357.416,E2 20357.416} C_VEL
LIN {X 0,Y 420.826,Z 373.806,A -85,B 0,C 180,E1 20355.857,E2 20355.857} C_VEL
LIN {X 0,Y 419.073,Z 371.165,A -85,B 0,C 180,E1 20354.897,E2 20354.897} C_VEL
LIN {X 0,Y 418.534,Z 369.058,A -85,B 0,C 180,E1 20354.461,E2 20354.461} C_VEL
LIN {X 0,Y 418.524,Z 369.067,A -85,B 0,C 180,E1 20350.601,E2 20350.601} C_VEL
LIN {X 0,Y 418.506,Z 369.102,A -85,B 0,C 180,E1 20346.861,E2 20346.861} C_VEL
LIN {X 0,Y 418.486,Z 369.072,A -85,B 0,C 180,E1 20343.15,E2 20343.15} C_VEL
LIN {X 0,Y 418.483,Z 369.059,A -85,B 0,C 180,E1 20339.315,E2 20339.315} C_VEL
LIN {X 0,Y 418.489,Z 369.078,A -85,B 0,C 180,E1 20335.478,E2 20335.478} C_VEL
LIN {X 0,Y 418.51,Z 369.095,A -85,B 0,C 180,E1 20331.758,E2 20331.758} C_VEL
LIN {X 0,Y 418.525,Z 369.06,A -85,B 0,C 180,E1 20328.004,E2 20328.004} C_VEL
LIN {X 0,Y 418.516,Z 369.061,A -85,B 0,C 180,E1 20324.327,E2 20324.327} C_VEL
LIN {X 0,Y 418.514,Z 369.269,A -85,B 0,C 180,E1 20323.071,E2 20323.071} C_VEL
LIN {X 0,Y 419.428,Z 371.93,A -85,B 0,C 180,E1 20322.473,E2 20322.473} C_VEL
LIN {X 0,Y 421.919,Z 374.717,A -85,B 0,C 180,E1 20321.198,E2 20321.198} C_VEL
LIN {X 0,Y 424.495,Z 375.974,A -85,B 0,C 180,E1 20320.065,E2 20320.065} C_VEL
LIN {X 0,Y 426.155,Z 379.317,A -85,B 0,C 180,E1 20319.25,E2 20319.25} C_VEL
LIN {X 0,Y 428.96,Z 381.799,A -85,B 0,C 180,E1 20318.102,E2 20318.102} C_VEL
LIN {X 0,Y 430.281,Z 382.728,A -85,B 0,C 180,E1 20317.598,E2 20317.598} C_VEL
LIN {X 0,Y 432.629,Z 386.398,A -85,B 0,C 180,E1 20316.648,E2 20316.648} C_VEL
LIN {X 0,Y 435.876,Z 389.234,A -85,B 0,C 180,E1 20315.503,E2 20315.503} C_VEL
LIN {X 0,Y 438.94,Z 393.394,A -85,B 0,C 180,E1 20314.426,E2 20314.426} C_VEL
LIN {X 0,Y 441.207,Z 395.549,A -85,B 0,C 180,E1 20313.701,E2 20313.701} C_VEL
LIN {X 0,Y 444.82,Z 400.05,A -85,B 0,C 180,E1 20312.56,E2 20312.56} C_VEL
LIN {X 0,Y 446.499,Z 401.996,A -85,B 0,C 180,E1 20312.057,E2 20312.057} C_VEL
LIN {X 0,Y 451.267,Z 407.869,A -85,B 0,C 180,E1 20310.68,E2 20310.68} C_VEL
LIN {X 0,Y 456.246,Z 414.141,A -85,B 0,C 180,E1 20309.33,E2 20309.33} C_VEL
LIN {X 0,Y 463.604,Z 423.42,A -85,B 0,C 180,E1 20307.481,E2 20307.481} C_VEL
LIN {X 0,Y 474.453,Z 438.155,A -85,B 0,C 180,E1 20304.987,E2 20304.987} C_VEL
LIN {X 0,Y 486.127,Z 454.989,A -85,B 0,C 180,E1 20302.562,E2 20302.562} C_VEL
LIN {X 0,Y 497.481,Z 472.781,A -85,B 0,C 180,E1 20300.399,E2 20300.399} C_VEL
LIN {X 0,Y 494.764,Z 530.037,A -85,B 0,C 180,E1 20299.492,E2 20299.492} C_VEL
LIN {X 0,Y 484.411,Z 743.234,A -85,B 0,C 180,E1 20296.161,E2 20296.161} C_VEL
LIN {X 0,Y 481.987,Z 769.926,A -85,B 0,C 180,E1 20295.568,E2 20295.568} C_VEL
LIN {X 0,Y 479.3,Z 791.582,A -85,B 0,C 180,E1 20294.913,E2 20294.913} C_VEL
LIN {X 0,Y 475.451,Z 816.4,A -85,B 0,C 180,E1 20293.948,E2 20293.948} C_VEL
LIN {X 0,Y 471.704,Z 836.768,A -85,B 0,C 180,E1 20292.961,E2 20292.961} C_VEL
LIN {X 0,Y 466.993,Z 859.147,A -85,B 0,C 180,E1 20291.668,E2 20291.668} C_VEL
LIN {X 0,Y 462.092,Z 879.669,A -85,B 0,C 180,E1 20290.233,E2 20290.233} C_VEL
LIN {X 0,Y 456.702,Z 900.554,A -85,B 0,C 180,E1 20288.526,E2 20288.526} C_VEL
LIN {X 0,Y 451.337,Z 919.524,A -85,B 0,C 180,E1 20286.681,E2 20286.681} C_VEL
LIN {X 0,Y 446.028,Z 937.684,A -85,B 0,C 180,E1 20284.641,E2 20284.641} C_VEL
LIN {X 0,Y 440.715,Z 954.826,A -85,B 0,C 180,E1 20282.373,E2 20282.373} C_VEL
LIN {X 0,Y 436.139,Z 969.53,A -85,B 0,C 180,E1 20280.138,E2 20280.138} C_VEL
LIN {X 0,Y 431.22,Z 985.321,A -85,B 0,C 180,E1 20277.33,E2 20277.33} C_VEL
LIN {X 0,Y 427.607,Z 997.226,A -85,B 0,C 180,E1 20274.868,E2 20274.868} C_VEL
LIN {X 0,Y 423.882,Z 1010.18,A -85,B 0,C 180,E1 20271.737,E2 20271.737} C_VEL
LIN {X 0,Y 421.31,Z 1019.806,A -85,B 0,C 180,E1 20268.974,E2 20268.974} C_VEL
LIN {X 0,Y 419.123,Z 1029.244,A -85,B 0,C 180,E1 20265.781,E2 20265.781} C_VEL
LIN {X 0,Y 417.622,Z 1036.803,A -85,B 0,C 180,E1 20262.584,E2 20262.584} C_VEL
LIN {X 0,Y 416.736,Z 1042.66,A -85,B 0,C 180,E1 20259.529,E2 20259.529} C_VEL
LIN {X 0,Y 416.211,Z 1047.36,A -85,B 0,C 180,E1 20256.206,E2 20256.206} C_VEL
LIN {X 0,Y 416.029,Z 1050.081,A -85,B 0,C 180,E1 20253.445,E2 20253.445} C_VEL
LIN {X 0,Y 415.964,Z 1051.822,A -85,B 0,C 180,E1 20250.551,E2 20250.551} C_VEL
LIN {X 0,Y 415.945,Z 1052.314,A -85,B 0,C 180,E1 20248.413,E2 20248.413} C_VEL
LIN {X 0,Y 414.951,Z 1052.399,A -85,B 0,C 180,E1 20247.352,E2 20247.352} C_VEL
LIN {X 0,Y 408.628,Z 1051.776,A -85,B 0,C 180,E1 20244.44,E2 20244.44} C_VEL
LIN {X 0,Y 408.018,Z 1051.383,A -85,B 0,C 180,E1 20243.583,E2 20243.583} C_VEL
LIN {X 0,Y 408.201,Z 1048.616,A -85,B 0,C 180,E1 20240.127,E2 20240.127} C_VEL
LIN {X 0,Y 408.619,Z 1044.904,A -85,B 0,C 180,E1 20237.134,E2 20237.134} C_VEL
LIN {X 0,Y 409.527,Z 1039.483,A -85,B 0,C 180,E1 20233.839,E2 20233.839} C_VEL
LIN {X 0,Y 411.021,Z 1032.276,A -85,B 0,C 180,E1 20230.532,E2 20230.532} C_VEL
LIN {X 0,Y 413.044,Z 1024.314,A -85,B 0,C 180,E1 20227.512,E2 20227.512} C_VEL
LIN {X 0,Y 416.061,Z 1013.749,A -85,B 0,C 180,E1 20224.216,E2 20224.216} C_VEL
LIN {X 0,Y 419.272,Z 1003.511,A -85,B 0,C 180,E1 20221.513,E2 20221.513} C_VEL
LIN {X 0,Y 423.933,Z 989.517,A -85,B 0,C 180,E1 20218.371,E2 20218.371} C_VEL
LIN {X 0,Y 428.3,Z 976.696,A -85,B 0,C 180,E1 20215.924,E2 20215.924} C_VEL
LIN {X 0,Y 433.702,Z 961.072,A -85,B 0,C 180,E1 20213.336,E2 20213.336} C_VEL
LIN {X 0,Y 439.234,Z 944.626,A -85,B 0,C 180,E1 20211.032,E2 20211.032} C_VEL
LIN {X 0,Y 445.194,Z 926.627,A -85,B 0,C 180,E1 20208.847,E2 20208.847} C_VEL
LIN {X 0,Y 450.958,Z 907.89,A -85,B 0,C 180,E1 20206.928,E2 20206.928} C_VEL
LIN {X 0,Y 456.331,Z 889.523,A -85,B 0,C 180,E1 20205.303,E2 20205.303} C_VEL
LIN {X 0,Y 461.985,Z 868.244,A -85,B 0,C 180,E1 20203.707,E2 20203.707} C_VEL
LIN {X 0,Y 466.58,Z 849.267,A -85,B 0,C 180,E1 20202.507,E2 20202.507} C_VEL
LIN {X 0,Y 471.476,Z 826.43,A -85,B 0,C 180,E1 20201.288,E2 20201.288} C_VEL
LIN {X 0,Y 475.423,Z 804.541,A -85,B 0,C 180,E1 20200.347,E2 20200.347} C_VEL
LIN {X 0,Y 478.794,Z 782.599,A -85,B 0,C 180,E1 20199.584,E2 20199.584} C_VEL
LIN {X 0,Y 481.612,Z 758.204,A -85,B 0,C 180,E1 20198.943,E2 20198.943} C_VEL
LIN {X 0,Y 483.399,Z 735.99,A -85,B 0,C 180,E1 20198.512,E2 20198.512} C_VEL
LIN {X 0,Y 496.612,Z 485.407,A -85,B 0,C 180,E1 20194.598,E2 20194.598} C_VEL
LIN {X 0,Y 496.914,Z 479.493,A -85,B 0,C 180,E1 20194.502,E2 20194.502} C_VEL
LIN {X 0,Y 486.438,Z 463.357,A -85,B 0,C 180,E1 20192.306,E2 20192.306} C_VEL
LIN {X 0,Y 476.625,Z 449.248,A -85,B 0,C 180,E1 20190.057,E2 20190.057} C_VEL
LIN {X 0,Y 466.885,Z 436.027,A -85,B 0,C 180,E1 20187.589,E2 20187.589} C_VEL
LIN {X 0,Y 458.438,Z 425.238,A -85,B 0,C 180,E1 20185.205,E2 20185.205} C_VEL
LIN {X 0,Y 454.01,Z 419.728,A -85,B 0,C 180,E1 20183.837,E2 20183.837} C_VEL
LIN {X 0,Y 449.722,Z 414.447,A -85,B 0,C 180,E1 20182.415,E2 20182.415} C_VEL
LIN {X 0,Y 446.007,Z 409.892,A -85,B 0,C 180,E1 20181.089,E2 20181.089} C_VEL
LIN {X 0,Y 441.392,Z 404.67,A -85,B 0,C 180,E1 20179.314,E2 20179.314} C_VEL
LIN {X 0,Y 440.218,Z 403.028,A -85,B 0,C 180,E1 20178.816,E2 20178.816} C_VEL
LIN {X 0,Y 436.857,Z 399.787,A -85,B 0,C 180,E1 20177.379,E2 20177.379} C_VEL
LIN {X 0,Y 435.195,Z 396.978,A -85,B 0,C 180,E1 20176.553,E2 20176.553} C_VEL
LIN {X 0,Y 431.677,Z 394.181,A -85,B 0,C 180,E1 20174.83,E2 20174.83} C_VEL
LIN {X 0,Y 429.405,Z 390.424,A -85,B 0,C 180,E1 20173.465,E2 20173.465} C_VEL
LIN {X 0,Y 426.191,Z 388.334,A -85,B 0,C 180,E1 20171.503,E2 20171.503} C_VEL
LIN {X 0,Y 424.238,Z 385.362,A -85,B 0,C 180,E1 20169.976,E2 20169.976} C_VEL
LIN {X 0,Y 423.604,Z 383.808,A -85,B 0,C 180,E1 20169.374,E2 20169.374} C_VEL
LIN {X 0,Y 419.601,Z 381.497,A -85,B 0,C 180,E1 20165.333,E2 20165.333} C_VEL
LIN {X 0,Y 417.71,Z 378.085,A -85,B 0,C 180,E1 20160.549,E2 20160.549} C_VEL
LIN {X 0,Y 417.634,Z 377.717,A -85,B 0,C 180,E1 20159.04,E2 20159.04} C_VEL
LIN {X 0,Y 417.839,Z 378.527,A -85,B 0,C 180,E1 20156.982,E2 20156.982} C_VEL
LIN {X 0,Y 422.288,Z 383.391,A -85,B 0,C 180,E1 20150.046,E2 20150.046} C_VEL
LIN {X 0,Y 423.813,Z 384.126,A -85,B 0,C 180,E1 20148.776,E2 20148.776} C_VEL
LIN {X 0,Y 425.701,Z 387.832,A -85,B 0,C 180,E1 20147.176,E2 20147.176} C_VEL
LIN {X 0,Y 429.146,Z 390.329,A -85,B 0,C 180,E1 20145.011,E2 20145.011} C_VEL
LIN {X 0,Y 429.818,Z 390.941,A -85,B 0,C 180,E1 20144.621,E2 20144.621} C_VEL
LIN {X 0,Y 432.013,Z 394.604,A -85,B 0,C 180,E1 20143.322,E2 20143.322} C_VEL
LIN {X 0,Y 435.424,Z 397.4,A -85,B 0,C 180,E1 20141.663,E2 20141.663} C_VEL
LIN {X 0,Y 438.244,Z 401.378,A -85,B 0,C 180,E1 20140.334,E2 20140.334} C_VEL
LIN {X 0,Y 440.955,Z 403.845,A -85,B 0,C 180,E1 20139.214,E2 20139.214} C_VEL
LIN {X 0,Y 444.176,Z 408.061,A -85,B 0,C 180,E1 20137.918,E2 20137.918} C_VEL
LIN {X 0,Y 446.477,Z 410.615,A -85,B 0,C 180,E1 20137.066,E2 20137.066} C_VEL
LIN {X 0,Y 453.195,Z 419.578,A -85,B 0,C 180,E1 20134.728,E2 20134.728} C_VEL
LIN {X 0,Y 460.636,Z 429.689,A -85,B 0,C 180,E1 20132.426,E2 20132.426} C_VEL
LIN {X 0,Y 470.755,Z 444.426,A -85,B 0,C 180,E1 20129.634,E2 20129.634} C_VEL
LIN {X 0,Y 479.537,Z 458.096,A -85,B 0,C 180,E1 20127.455,E2 20127.455} C_VEL
LIN {X 0,Y 489.467,Z 474.407,A -85,B 0,C 180,E1 20125.206,E2 20125.206} C_VEL
LIN {X 0,Y 496.703,Z 487.414,A -85,B 0,C 180,E1 20123.673,E2 20123.673} C_VEL
LIN {X 0,Y 483.715,Z 735.877,A -85,B 0,C 180,E1 20119.794,E2 20119.794} C_VEL
LIN {X 0,Y 481.585,Z 768.891,A -85,B 0,C 180,E1 20119.228,E2 20119.228} C_VEL
LIN {X 0,Y 479.113,Z 790.852,A -85,B 0,C 180,E1 20118.715,E2 20118.715} C_VEL
LIN {X 0,Y 475.675,Z 814.589,A -85,B 0,C 180,E1 20117.994,E2 20117.994} C_VEL
LIN {X 0,Y 471.623,Z 836.841,A -85,B 0,C 180,E1 20117.113,E2 20117.113} C_VEL
LIN {X 0,Y 467.194,Z 858.258,A -85,B 0,C 180,E1 20116.078,E2 20116.078} C_VEL
LIN {X 0,Y 461.758,Z 881.059,A -85,B 0,C 180,E1 20114.729,E2 20114.729} C_VEL
LIN {X 0,Y 456.832,Z 899.811,A -85,B 0,C 180,E1 20113.414,E2 20113.414} C_VEL
LIN {X 0,Y 450.533,Z 921.941,A -85,B 0,C 180,E1 20111.574,E2 20111.574} C_VEL
LIN {X 0,Y 445.236,Z 939.264,A -85,B 0,C 180,E1 20109.879,E2 20109.879} C_VEL
LIN {X 0,Y 439.281,Z 958.022,A -85,B 0,C 180,E1 20107.756,E2 20107.756} C_VEL
LIN {X 0,Y 433.72,Z 974.787,A -85,B 0,C 180,E1 20105.518,E2 20105.518} C_VEL
LIN {X 0,Y 428.26,Z 991.425,A -85,B 0,C 180,E1 20102.956,E2 20102.956} C_VEL
LIN {X 0,Y 423.261,Z 1006.471,A -85,B 0,C 180,E1 20100.211,E2 20100.211} C_VEL
LIN {X 0,Y 418.917,Z 1020.369,A -85,B 0,C 180,E1 20097.276,E2 20097.276} C_VEL
LIN {X 0,Y 415.238,Z 1032.683,A -85,B 0,C 180,E1 20094.165,E2 20094.165} C_VEL
LIN {X 0,Y 412.463,Z 1043.321,A -85,B 0,C 180,E1 20091.025,E2 20091.025} C_VEL
LIN {X 0,Y 410.374,Z 1052.541,A -85,B 0,C 180,E1 20087.694,E2 20087.694} C_VEL
LIN {X 0,Y 409.108,Z 1059.679,A -85,B 0,C 180,E1 20084.58,E2 20084.58} C_VEL
LIN {X 0,Y 408.324,Z 1065.806,A -85,B 0,C 180,E1 20081.154,E2 20081.154} C_VEL
LIN {X 0,Y 408.032,Z 1069.618,A -85,B 0,C 180,E1 20078.313,E2 20078.313} C_VEL
LIN {X 0,Y 407.95,Z 1072.436,A -85,B 0,C 180,E1 20075.344,E2 20075.344} C_VEL
LIN {X 0,Y 407.948,Z 1074.103,A -85,B 0,C 180,E1 20071.966,E2 20071.966} C_VEL
LIN {X 0,Y 407.956,Z 1074.241,A -85,B 0,C 180,E1 20069.157,E2 20069.157} C_VEL
LIN {X 0,Y 407.948,Z 1073.363,A -85,B 0,C 180,E1 20066.487,E2 20066.487} C_VEL
LIN {X 0,Y 407.961,Z 1071.137,A -85,B 0,C 180,E1 20063.385,E2 20063.385} C_VEL
LIN {X 0,Y 408.167,Z 1067.01,A -85,B 0,C 180,E1 20059.984,E2 20059.984} C_VEL
LIN {X 0,Y 408.624,Z 1062.315,A -85,B 0,C 180,E1 20057.134,E2 20057.134} C_VEL
LIN {X 0,Y 409.629,Z 1055.477,A -85,B 0,C 180,E1 20053.843,E2 20053.843} C_VEL
LIN {X 0,Y 411.236,Z 1047.009,A -85,B 0,C 180,E1 20050.63,E2 20050.63} C_VEL
LIN {X 0,Y 413.622,Z 1036.878,A -85,B 0,C 180,E1 20047.396,E2 20047.396} C_VEL
LIN {X 0,Y 416.776,Z 1024.965,A -85,B 0,C 180,E1 20044.263,E2 20044.263} C_VEL
LIN {X 0,Y 420.625,Z 1011.871,A -85,B 0,C 180,E1 20041.303,E2 20041.303} C_VEL
LIN {X 0,Y 425.062,Z 997.252,A -85,B 0,C 180,E1 20038.519,E2 20038.519} C_VEL
LIN {X 0,Y 429.759,Z 982.357,A -85,B 0,C 180,E1 20036.055,E2 20036.055} C_VEL
LIN {X 0,Y 435.272,Z 964.751,A -85,B 0,C 180,E1 20033.572,E2 20033.572} C_VEL
LIN {X 0,Y 440.316,Z 948.391,A -85,B 0,C 180,E1 20031.577,E2 20031.577} C_VEL
LIN {X 0,Y 446.532,Z 927.33,A -85,B 0,C 180,E1 20029.385,E2 20029.385} C_VEL
LIN {X 0,Y 451.536,Z 909.429,A -85,B 0,C 180,E1 20027.798,E2 20027.798} C_VEL
LIN {X 0,Y 457.42,Z 886.738,A -85,B 0,C 180,E1 20026.089,E2 20026.089} C_VEL
LIN {X 0,Y 462.003,Z 867.268,A -85,B 0,C 180,E1 20024.863,E2 20024.863} C_VEL
LIN {X 0,Y 466.68,Z 845.234,A -85,B 0,C 180,E1 20023.688,E2 20023.688} C_VEL
LIN {X 0,Y 470.806,Z 822.209,A -85,B 0,C 180,E1 20022.707,E2 20022.707} C_VEL
LIN {X 0,Y 474.445,Z 798.599,A -85,B 0,C 180,E1 20021.903,E2 20021.903} C_VEL
LIN {X 0,Y 477.272,Z 774.156,A -85,B 0,C 180,E1 20021.29,E2 20021.29} C_VEL
LIN {X 0,Y 479.108,Z 750.268,A -85,B 0,C 180,E1 20020.838,E2 20020.838} C_VEL
LIN {X 0,Y 491.484,Z 500.014,A -85,B 0,C 180,E1 20016.927,E2 20016.927} C_VEL
LIN {X 0,Y 492.133,Z 484.433,A -85,B 0,C 180,E1 20016.661,E2 20016.661} C_VEL
LIN {X 0,Y 481.223,Z 465.091,A -85,B 0,C 180,E1 20014.468,E2 20014.468} C_VEL
LIN {X 0,Y 471.922,Z 449.921,A -85,B 0,C 180,E1 20012.451,E2 20012.451} C_VEL
LIN {X 0,Y 462.572,Z 435.394,A -85,B 0,C 180,E1 20010.242,E2 20010.242} C_VEL
LIN {X 0,Y 452.69,Z 421.179,A -85,B 0,C 180,E1 20007.671,E2 20007.671} C_VEL
LIN {X 0,Y 444.329,Z 409.768,A -85,B 0,C 180,E1 20005.242,E2 20005.242} C_VEL
LIN {X 0,Y 438.133,Z 401.889,A -85,B 0,C 180,E1 20003.254,E2 20003.254} C_VEL
LIN {X 0,Y 434.632,Z 398.042,A -85,B 0,C 180,E1 20002.059,E2 20002.059} C_VEL
LIN {X 0,Y 433.205,Z 396.022,A -85,B 0,C 180,E1 20001.53,E2 20001.53} C_VEL
LIN {X 0,Y 429.823,Z 392.754,A -85,B 0,C 180,E1 20000.281,E2 20000.281} C_VEL
LIN {X 0,Y 427.998,Z 389.885,A -85,B 0,C 180,E1 19999.517,E2 19999.517} C_VEL
LIN {X 0,Y 424.721,Z 387.166,A -85,B 0,C 180,E1 19998.176,E2 19998.176} C_VEL
LIN {X 0,Y 422.415,Z 383.477,A -85,B 0,C 180,E1 19997.069,E2 19997.069} C_VEL
LIN {X 0,Y 418.953,Z 381.085,A -85,B 0,C 180,E1 19995.433,E2 19995.433} C_VEL
LIN {X 0,Y 417.166,Z 378.034,A -85,B 0,C 180,E1 19994.399,E2 19994.399} C_VEL
LIN {X 0,Y 416.708,Z 376.859,A -85,B 0,C 180,E1 19994.096,E2 19994.096} C_VEL
LIN {X 0,Y 413.117,Z 375.015,A -85,B 0,C 180,E1 19992.014,E2 19992.014} C_VEL
LIN {X 0,Y 411.261,Z 372.43,A -85,B 0,C 180,E1 19990.648,E2 19990.648} C_VEL
LIN {X 0,Y 410.558,Z 370.05,A -85,B 0,C 180,E1 19989.957,E2 19989.957} C_VEL
LIN {X 0,Y 410.581,Z 370.069,A -85,B 0,C 180,E1 19986.151,E2 19986.151} C_VEL
LIN {X 0,Y 410.588,Z 370.079,A -85,B 0,C 180,E1 19982.233,E2 19982.233} C_VEL
LIN {X 0,Y 410.584,Z 370.046,A -85,B 0,C 180,E1 19978.465,E2 19978.465} C_VEL
LIN {X 0,Y 410.561,Z 370.05,A -85,B 0,C 180,E1 19974.69,E2 19974.69} C_VEL
LIN {X 0,Y 410.552,Z 370.081,A -85,B 0,C 180,E1 19970.891,E2 19970.891} C_VEL
LIN {X 0,Y 410.586,Z 370.24,A -85,B 0,C 180,E1 19967.586,E2 19967.586} C_VEL
LIN {X 0,Y 411.424,Z 372.836,A -85,B 0,C 180,E1 19966.794,E2 19966.794} C_VEL
LIN {X 0,Y 413.977,Z 375.683,A -85,B 0,C 180,E1 19965.022,E2 19965.022} C_VEL
LIN {X 0,Y 416.823,Z 377.106,A -85,B 0,C 180,E1 19963.413,E2 19963.413} C_VEL
LIN {X 0,Y 418.358,Z 380.281,A -85,B 0,C 180,E1 19962.474,E2 19962.474} C_VEL
LIN {X 0,Y 420.981,Z 382.788,A -85,B 0,C 180,E1 19961.154,E2 19961.154} C_VEL
LIN {X 0,Y 422.785,Z 383.886,A -85,B 0,C 180,E1 19960.341,E2 19960.341} C_VEL
LIN {X 0,Y 424.891,Z 387.415,A -85,B 0,C 180,E1 19959.329,E2 19959.329} C_VEL
LIN {X 0,Y 428.425,Z 390.389,A -85,B 0,C 180,E1 19957.893,E2 19957.893} C_VEL
LIN {X 0,Y 431.175,Z 394.303,A -85,B 0,C 180,E1 19956.782,E2 19956.782} C_VEL
LIN {X 0,Y 433.863,Z 396.716,A -85,B 0,C 180,E1 19955.817,E2 19955.817} C_VEL
LIN {X 0,Y 437.263,Z 401.125,A -85,B 0,C 180,E1 19954.611,E2 19954.611} C_VEL
LIN {X 0,Y 439.121,Z 403.021,A -85,B 0,C 180,E1 19954.003,E2 19954.003} C_VEL
LIN {X 0,Y 442.898,Z 407.603,A -85,B 0,C 180,E1 19952.795,E2 19952.795} C_VEL
LIN {X 0,Y 448.961,Z 415.194,A -85,B 0,C 180,E1 19950.99,E2 19950.99} C_VEL
LIN {X 0,Y 453.778,Z 421.318,A -85,B 0,C 180,E1 19949.659,E2 19949.659} C_VEL
LIN {X 0,Y 461.047,Z 430.651,A -85,B 0,C 180,E1 19947.794,E2 19947.794} C_VEL
LIN {X 0,Y 471.423,Z 444.915,A -85,B 0,C 180,E1 19945.359,E2 19945.359} C_VEL
LIN {X 0,Y 482.75,Z 461.466,A -85,B 0,C 180,E1 19942.953,E2 19942.953} C_VEL
LIN {X 0,Y 492.491,Z 476.891,A -85,B 0,C 180,E1 19941.044,E2 19941.044} C_VEL
LIN {X 0,Y 479.792,Z 731.368,A -85,B 0,C 180,E1 19937.074,E2 19937.074} C_VEL
LIN {X 0,Y 477.984,Z 756.062,A -85,B 0,C 180,E1 19936.608,E2 19936.608} C_VEL
LIN {X 0,Y 475.502,Z 779.25,A -85,B 0,C 180,E1 19936.015,E2 19936.015} C_VEL
LIN {X 0,Y 472.191,Z 802.335,A -85,B 0,C 180,E1 19935.228,E2 19935.228} C_VEL
LIN {X 0,Y 468.813,Z 822.107,A -85,B 0,C 180,E1 19934.392,E2 19934.392} C_VEL
LIN {X 0,Y 464.329,Z 844.943,A -85,B 0,C 180,E1 19933.219,E2 19933.219} C_VEL
LIN {X 0,Y 459.73,Z 864.986,A -85,B 0,C 180,E1 19931.974,E2 19931.974} C_VEL
LIN {X 0,Y 454.482,Z 886.14,A -85,B 0,C 180,E1 19930.427,E2 19930.427} C_VEL
LIN {X 0,Y 449.076,Z 905.598,A -85,B 0,C 180,E1 19928.731,E2 19928.731} C_VEL
LIN {X 0,Y 443.95,Z 923.103,A -85,B 0,C 180,E1 19926.967,E2 19926.967} C_VEL
LIN {X 0,Y 437.883,Z 942.682,A -85,B 0,C 180,E1 19924.651,E2 19924.651} C_VEL
LIN {X 0,Y 432.985,Z 957.931,A -85,B 0,C 180,E1 19922.552,E2 19922.552} C_VEL
LIN {X 0,Y 427.321,Z 975.393,A -85,B 0,C 180,E1 19919.74,E2 19919.74} C_VEL
LIN {X 0,Y 423.112,Z 988.41,A -85,B 0,C 180,E1 19917.288,E2 19917.288} C_VEL
LIN {X 0,Y 418.604,Z 1002.813,A -85,B 0,C 180,E1 19914.108,E2 19914.108} C_VEL
LIN {X 0,Y 415.435,Z 1013.514,A -85,B 0,C 180,E1 19911.311,E2 19911.311} C_VEL
LIN {X 0,Y 412.531,Z 1024.412,A -85,B 0,C 180,E1 19907.928,E2 19907.928} C_VEL
LIN {X 0,Y 410.692,Z 1032.286,A -85,B 0,C 180,E1 19904.956,E2 19904.956} C_VEL
LIN {X 0,Y 409.303,Z 1039.625,A -85,B 0,C 180,E1 19901.589,E2 19901.589} C_VEL
LIN {X 0,Y 408.523,Z 1044.83,A -85,B 0,C 180,E1 19898.445,E2 19898.445} C_VEL
LIN {X 0,Y 408.159,Z 1048.539,A -85,B 0,C 180,E1 19895.482,E2 19895.482} C_VEL
LIN {X 0,Y 407.999,Z 1051.38,A -85,B 0,C 180,E1 19891.966,E2 19891.966} C_VEL
LIN {X 0,Y 407.964,Z 1052.407,A -85,B 0,C 180,E1 19889.157,E2 19889.157} C_VEL
LIN {X 0,Y 407.96,Z 1052.4,A -85,B 0,C 180,E1 19886.346,E2 19886.346} C_VEL
LIN {X 0,Y 408.018,Z 1051.383,A -85,B 0,C 180,E1 19883.583,E2 19883.583} C_VEL
LIN {X 0,Y 407.067,Z 1050.788,A -85,B 0,C 180,E1 19882.504,E2 19882.504} C_VEL
LIN {X 0,Y 400.81,Z 1048.289,A -85,B 0,C 180,E1 19879.47,E2 19879.47} C_VEL
LIN {X 0,Y 400.372,Z 1047.462,A -85,B 0,C 180,E1 19878.682,E2 19878.682} C_VEL
LIN {X 0,Y 401.121,Z 1042.412,A -85,B 0,C 180,E1 19875.123,E2 19875.123} C_VEL
LIN {X 0,Y 402.193,Z 1036.974,A -85,B 0,C 180,E1 19872.194,E2 19872.194} C_VEL
LIN {X 0,Y 404.102,Z 1029.272,A -85,B 0,C 180,E1 19868.823,E2 19868.823} C_VEL
LIN {X 0,Y 406.684,Z 1020.075,A -85,B 0,C 180,E1 19865.603,E2 19865.603} C_VEL
LIN {X 0,Y 410.136,Z 1009.29,A -85,B 0,C 180,E1 19862.406,E2 19862.406} C_VEL
LIN {X 0,Y 414.282,Z 997.002,A -85,B 0,C 180,E1 19859.386,E2 19859.386} C_VEL
LIN {X 0,Y 418.81,Z 984.227,A -85,B 0,C 180,E1 19856.68,E2 19856.68} C_VEL
LIN {X 0,Y 424.332,Z 968.783,A -85,B 0,C 180,E1 19853.907,E2 19853.907} C_VEL
LIN {X 0,Y 429.412,Z 954.485,A -85,B 0,C 180,E1 19851.694,E2 19851.694} C_VEL
LIN {X 0,Y 435.981,Z 935.537,A -85,B 0,C 180,E1 19849.184,E2 19849.184} C_VEL
LIN {X 0,Y 441.536,Z 918.763,A -85,B 0,C 180,E1 19847.294,E2 19847.294} C_VEL
LIN {X 0,Y 447.949,Z 898.327,A -85,B 0,C 180,E1 19845.322,E2 19845.322} C_VEL
LIN {X 0,Y 453.407,Z 879.276,A -85,B 0,C 180,E1 19843.769,E2 19843.769} C_VEL
LIN {X 0,Y 458.932,Z 858.441,A -85,B 0,C 180,E1 19842.317,E2 19842.317} C_VEL
LIN {X 0,Y 464.038,Z 836.256,A -85,B 0,C 180,E1 19841.047,E2 19841.047} C_VEL
LIN {X 0,Y 468.264,Z 815.417,A -85,B 0,C 180,E1 19840.048,E2 19840.048} C_VEL
LIN {X 0,Y 472.296,Z 791.455,A -85,B 0,C 180,E1 19839.13,E2 19839.13} C_VEL
LIN {X 0,Y 475.196,Z 770.065,A -85,B 0,C 180,E1 19838.487,E2 19838.487} C_VEL
LIN {X 0,Y 477.824,Z 743.477,A -85,B 0,C 180,E1 19837.901,E2 19837.901} C_VEL
LIN {X 0,Y 490.203,Z 517.058,A -85,B 0,C 180,E1 19834.329,E2 19834.329} C_VEL
LIN {X 0,Y 491.989,Z 483.415,A -85,B 0,C 180,E1 19833.787,E2 19833.787} C_VEL
LIN {X 0,Y 480.98,Z 466.388,A -85,B 0,C 180,E1 19831.383,E2 19831.383} C_VEL
LIN {X 0,Y 471.213,Z 452.45,A -85,B 0,C 180,E1 19829.039,E2 19829.039} C_VEL
LIN {X 0,Y 463.001,Z 441.37,A -85,B 0,C 180,E1 19826.865,E2 19826.865} C_VEL
LIN {X 0,Y 455.92,Z 432.167,A -85,B 0,C 180,E1 19824.799,E2 19824.799} C_VEL
LIN {X 0,Y 451.75,Z 426.891,A -85,B 0,C 180,E1 19823.479,E2 19823.479} C_VEL
LIN {X 0,Y 447.528,Z 421.652,A -85,B 0,C 180,E1 19822.046,E2 19822.046} C_VEL
LIN {X 0,Y 443.072,Z 416.189,A -85,B 0,C 180,E1 19820.406,E2 19820.406} C_VEL
LIN {X 0,Y 439.439,Z 411.92,A -85,B 0,C 180,E1 19818.954,E2 19818.954} C_VEL
LIN {X 0,Y 438.344,Z 410.514,A -85,B 0,C 180,E1 19818.486,E2 19818.486} C_VEL
LIN {X 0,Y 434.931,Z 406.953,A -85,B 0,C 180,E1 19816.976,E2 19816.976} C_VEL
LIN {X 0,Y 433.411,Z 404.566,A -85,B 0,C 180,E1 19816.21,E2 19816.21} C_VEL
LIN {X 0,Y 429.882,Z 401.428,A -85,B 0,C 180,E1 19814.411,E2 19814.411} C_VEL
LIN {X 0,Y 427.982,Z 398.219,A -85,B 0,C 180,E1 19813.236,E2 19813.236} C_VEL
LIN {X 0,Y 424.655,Z 395.833,A -85,B 0,C 180,E1 19811.132,E2 19811.132} C_VEL
LIN {X 0,Y 422.725,Z 392.54,A -85,B 0,C 180,E1 19809.531,E2 19809.531} C_VEL
LIN {X 0,Y 422.299,Z 391.674,A -85,B 0,C 180,E1 19809.128,E2 19809.128} C_VEL
LIN {X 0,Y 418.26,Z 389.093,A -85,B 0,C 180,E1 19804.8,E2 19804.8} C_VEL
LIN {X 0,Y 416.718,Z 385.975,A -85,B 0,C 180,E1 19800.412,E2 19800.412} C_VEL
LIN {X 0,Y 416.659,Z 385.66,A -85,B 0,C 180,E1 19799.037,E2 19799.037} C_VEL
LIN {X 0,Y 416.861,Z 386.506,A -85,B 0,C 180,E1 19796.975,E2 19796.975} C_VEL
LIN {X 0,Y 421.336,Z 391.347,A -85,B 0,C 180,E1 19790.015,E2 19790.015} C_VEL
LIN {X 0,Y 422.519,Z 391.901,A -85,B 0,C 180,E1 19789.018,E2 19789.018} C_VEL
LIN {X 0,Y 424.546,Z 395.749,A -85,B 0,C 180,E1 19787.278,E2 19787.278} C_VEL
LIN {X 0,Y 428.342,Z 398.664,A -85,B 0,C 180,E1 19784.879,E2 19784.879} C_VEL
LIN {X 0,Y 430.683,Z 402.432,A -85,B 0,C 180,E1 19783.477,E2 19783.477} C_VEL
LIN {X 0,Y 433.847,Z 405.141,A -85,B 0,C 180,E1 19781.907,E2 19781.907} C_VEL
LIN {X 0,Y 436.854,Z 409.216,A -85,B 0,C 180,E1 19780.478,E2 19780.478} C_VEL
LIN {X 0,Y 439.157,Z 411.365,A -85,B 0,C 180,E1 19779.509,E2 19779.509} C_VEL
LIN {X 0,Y 442.576,Z 415.762,A -85,B 0,C 180,E1 19778.113,E2 19778.113} C_VEL
LIN {X 0,Y 444.917,Z 418.595,A -85,B 0,C 180,E1 19777.225,E2 19777.225} C_VEL
LIN {X 0,Y 450.958,Z 426.734,A -85,B 0,C 180,E1 19775.085,E2 19775.085} C_VEL
LIN {X 0,Y 458.382,Z 436.992,A -85,B 0,C 180,E1 19772.736,E2 19772.736} C_VEL
LIN {X 0,Y 468.267,Z 451.648,A -85,B 0,C 180,E1 19769.952,E2 19769.952} C_VEL
LIN {X 0,Y 478.528,Z 467.841,A -85,B 0,C 180,E1 19767.378,E2 19767.378} C_VEL
LIN {X 0,Y 489.337,Z 486.411,A -85,B 0,C 180,E1 19764.922,E2 19764.922} C_VEL
LIN {X 0,Y 491.861,Z 491.26,A -85,B 0,C 180,E1 19764.372,E2 19764.372} C_VEL
LIN {X 0,Y 478.411,Z 740.602,A -85,B 0,C 180,E1 19760.46,E2 19760.46} C_VEL
LIN {X 0,Y 476.271,Z 770.622,A -85,B 0,C 180,E1 19759.928,E2 19759.928} C_VEL
LIN {X 0,Y 473.736,Z 792.208,A -85,B 0,C 180,E1 19759.415,E2 19759.415} C_VEL
LIN {X 0,Y 469.904,Z 817.136,A -85,B 0,C 180,E1 19758.632,E2 19758.632} C_VEL
LIN {X 0,Y 466.109,Z 837.319,A -85,B 0,C 180,E1 19757.821,E2 19757.821} C_VEL
LIN {X 0,Y 461.364,Z 859.57,A -85,B 0,C 180,E1 19756.735,E2 19756.735} C_VEL
LIN {X 0,Y 456.01,Z 881.169,A -85,B 0,C 180,E1 19755.439,E2 19755.439} C_VEL
LIN {X 0,Y 450.954,Z 899.799,A -85,B 0,C 180,E1 19754.125,E2 19754.125} C_VEL
LIN {X 0,Y 444.342,Z 922.247,A -85,B 0,C 180,E1 19752.239,E2 19752.239} C_VEL
LIN {X 0,Y 438.975,Z 939.213,A -85,B 0,C 180,E1 19750.563,E2 19750.563} C_VEL
LIN {X 0,Y 432.809,Z 957.929,A -85,B 0,C 180,E1 19748.422,E2 19748.422} C_VEL
LIN {X 0,Y 427.03,Z 974.683,A -85,B 0,C 180,E1 19746.161,E2 19746.161} C_VEL
LIN {X 0,Y 421.34,Z 991.304,A -85,B 0,C 180,E1 19743.569,E2 19743.569} C_VEL
LIN {X 0,Y 416.125,Z 1006.337,A -85,B 0,C 180,E1 19740.784,E2 19740.784} C_VEL
LIN {X 0,Y 411.569,Z 1020.223,A -85,B 0,C 180,E1 19737.804,E2 19737.804} C_VEL
LIN {X 0,Y 407.702,Z 1032.524,A -85,B 0,C 180,E1 19734.641,E2 19734.641} C_VEL
LIN {X 0,Y 404.684,Z 1043.503,A -85,B 0,C 180,E1 19731.331,E2 19731.331} C_VEL
LIN {X 0,Y 402.573,Z 1052.271,A -85,B 0,C 180,E1 19728.087,E2 19728.087} C_VEL
LIN {X 0,Y 401.249,Z 1059.188,A -85,B 0,C 180,E1 19725.02,E2 19725.02} C_VEL
LIN {X 0,Y 400.357,Z 1065.613,A -85,B 0,C 180,E1 19721.379,E2 19721.379} C_VEL
LIN {X 0,Y 400.047,Z 1069.421,A -85,B 0,C 180,E1 19718.48,E2 19718.48} C_VEL
LIN {X 0,Y 399.951,Z 1072.235,A -85,B 0,C 180,E1 19715.451,E2 19715.451} C_VEL
LIN {X 0,Y 399.951,Z 1073.892,A -85,B 0,C 180,E1 19712.006,E2 19712.006} C_VEL
LIN {X 0,Y 399.959,Z 1074.025,A -85,B 0,C 180,E1 19709.141,E2 19709.141} C_VEL
LIN {X 0,Y 399.948,Z 1073.142,A -85,B 0,C 180,E1 19706.417,E2 19706.417} C_VEL
LIN {X 0,Y 399.964,Z 1070.909,A -85,B 0,C 180,E1 19703.252,E2 19703.252} C_VEL
LIN {X 0,Y 400.185,Z 1066.77,A -85,B 0,C 180,E1 19699.782,E2 19699.782} C_VEL
LIN {X 0,Y 400.678,Z 1062.068,A -85,B 0,C 180,E1 19696.874,E2 19696.874} C_VEL
LIN {X 0,Y 401.756,Z 1055.217,A -85,B 0,C 180,E1 19693.518,E2 19693.518} C_VEL
LIN {X 0,Y 403.429,Z 1046.909,A -85,B 0,C 180,E1 19690.301,E2 19690.301} C_VEL
LIN {X 0,Y 405.86,Z 1037.07,A -85,B 0,C 180,E1 19687.092,E2 19687.092} C_VEL
LIN {X 0,Y 409.143,Z 1025.257,A -85,B 0,C 180,E1 19683.903,E2 19683.903} C_VEL
LIN {X 0,Y 412.928,Z 1012.863,A -85,B 0,C 180,E1 19681.034,E2 19681.034} C_VEL
LIN {X 0,Y 417.745,Z 997.718,A -85,B 0,C 180,E1 19678.064,E2 19678.064} C_VEL
LIN {X 0,Y 422.315,Z 983.746,A -85,B 0,C 180,E1 19675.702,E2 19675.702} C_VEL
LIN {X 0,Y 428.308,Z 965.43,A -85,B 0,C 180,E1 19673.049,E2 19673.049} C_VEL
LIN {X 0,Y 433.27,Z 949.908,A -85,B 0,C 180,E1 19671.118,E2 19671.118} C_VEL
LIN {X 0,Y 439.257,Z 930.606,A -85,B 0,C 180,E1 19669.036,E2 19669.036} C_VEL
LIN {X 0,Y 444.915,Z 911.03,A -85,B 0,C 180,E1 19667.257,E2 19667.257} C_VEL
LIN {X 0,Y 450.545,Z 890.396,A -85,B 0,C 180,E1 19665.647,E2 19665.647} C_VEL
LIN {X 0,Y 455.813,Z 868.823,A -85,B 0,C 180,E1 19664.256,E2 19664.256} C_VEL
LIN {X 0,Y 460.577,Z 847.137,A -85,B 0,C 180,E1 19663.078,E2 19663.078} C_VEL
LIN {X 0,Y 464.961,Z 823.854,A -85,B 0,C 180,E1 19662.059,E2 19662.059} C_VEL
LIN {X 0,Y 468.475,Z 801.857,A -85,B 0,C 180,E1 19661.291,E2 19661.291} C_VEL
LIN {X 0,Y 471.729,Z 775.805,A -85,B 0,C 180,E1 19660.608,E2 19660.608} C_VEL
LIN {X 0,Y 473.578,Z 753.395,A -85,B 0,C 180,E1 19660.172,E2 19660.172} C_VEL
LIN {X 0,Y 486.292,Z 505.518,A -85,B 0,C 180,E1 19656.269,E2 19656.269} C_VEL
LIN {X 0,Y 487.071,Z 488.034,A -85,B 0,C 180,E1 19655.972,E2 19655.972} C_VEL
LIN {X 0,Y 476.42,Z 469.074,A -85,B 0,C 180,E1 19653.755,E2 19653.755} C_VEL
LIN {X 0,Y 465.987,Z 451.929,A -85,B 0,C 180,E1 19651.391,E2 19651.391} C_VEL
LIN {X 0,Y 455.615,Z 436.082,A -85,B 0,C 180,E1 19648.798,E2 19648.798} C_VEL
LIN {X 0,Y 448.887,Z 426.559,A -85,B 0,C 180,E1 19646.955,E2 19646.955} C_VEL
LIN {X 0,Y 441.99,Z 416.9,A -85,B 0,C 180,E1 19644.884,E2 19644.884} C_VEL
LIN {X 0,Y 435.88,Z 409.12,A -85,B 0,C 180,E1 19642.882,E2 19642.882} C_VEL
LIN {X 0,Y 432.286,Z 404.919,A -85,B 0,C 180,E1 19641.614,E2 19641.614} C_VEL
LIN {X 0,Y 431.029,Z 403.342,A -85,B 0,C 180,E1 19641.145,E2 19641.145} C_VEL
LIN {X 0,Y 427.579,Z 399.663,A -85,B 0,C 180,E1 19639.821,E2 19639.821} C_VEL
LIN {X 0,Y 426.075,Z 397.406,A -85,B 0,C 180,E1 19639.181,E2 19639.181} C_VEL
LIN {X 0,Y 422.735,Z 394.337,A -85,B 0,C 180,E1 19637.766,E2 19637.766} C_VEL
LIN {X 0,Y 420.881,Z 391.233,A -85,B 0,C 180,E1 19636.848,E2 19636.848} C_VEL
LIN {X 0,Y 417.351,Z 388.627,A -85,B 0,C 180,E1 19635.138,E2 19635.138} C_VEL
LIN {X 0,Y 415.389,Z 385.174,A -85,B 0,C 180,E1 19633.964,E2 19633.964} C_VEL
LIN {X 0,Y 414.878,Z 384.579,A -85,B 0,C 180,E1 19633.662,E2 19633.662} C_VEL
LIN {X 0,Y 411.246,Z 382.217,A -85,B 0,C 180,E1 19631.429,E2 19631.429} C_VEL
LIN {X 0,Y 409.506,Z 379.103,A -85,B 0,C 180,E1 19630.019,E2 19630.019} C_VEL
LIN {X 0,Y 409.032,Z 377.905,A -85,B 0,C 180,E1 19629.569,E2 19629.569} C_VEL
LIN {X 0,Y 405.105,Z 375.919,A -85,B 0,C 180,E1 19625.808,E2 19625.808} C_VEL
LIN {X 0,Y 402.692,Z 371.474,A -85,B 0,C 180,E1 19619.858,E2 19619.858} C_VEL
LIN {X 0,Y 402.678,Z 371.328,A -85,B 0,C 180,E1 19618.008,E2 19618.008} C_VEL
LIN {X 0,Y 403.829,Z 374.366,A -85,B 0,C 180,E1 19613.745,E2 19613.745} C_VEL
LIN {X 0,Y 407.511,Z 377.451,A -85,B 0,C 180,E1 19609.253,E2 19609.253} C_VEL
LIN {X 0,Y 409.198,Z 378.17,A -85,B 0,C 180,E1 19607.869,E2 19607.869} C_VEL
LIN {X 0,Y 410.435,Z 381.109,A -85,B 0,C 180,E1 19606.762,E2 19606.762} C_VEL
LIN {X 0,Y 413.249,Z 383.839,A -85,B 0,C 180,E1 19604.852,E2 19604.852} C_VEL
LIN {X 0,Y 415.252,Z 384.872,A -85,B 0,C 180,E1 19603.709,E2 19603.709} C_VEL
LIN {X 0,Y 417.204,Z 388.397,A -85,B 0,C 180,E1 19602.528,E2 19602.528} C_VEL
LIN {X 0,Y 420.046,Z 390.833,A -85,B 0,C 180,E1 19601.111,E2 19601.111} C_VEL
LIN {X 0,Y 421.105,Z 391.631,A -85,B 0,C 180,E1 19600.62,E2 19600.62} C_VEL
LIN {X 0,Y 423.636,Z 395.448,A -85,B 0,C 180,E1 19599.41,E2 19599.41} C_VEL
LIN {X 0,Y 426.588,Z 397.977,A -85,B 0,C 180,E1 19598.191,E2 19598.191} C_VEL
LIN {X 0,Y 429.558,Z 402.02,A -85,B 0,C 180,E1 19596.98,E2 19596.98} C_VEL
LIN {X 0,Y 431.947,Z 404.299,A -85,B 0,C 180,E1 19596.103,E2 19596.103} C_VEL
LIN {X 0,Y 435.591,Z 408.847,A -85,B 0,C 180,E1 19594.798,E2 19594.798} C_VEL
LIN {X 0,Y 437.227,Z 410.734,A -85,B 0,C 180,E1 19594.246,E2 19594.246} C_VEL
LIN {X 0,Y 442.213,Z 416.886,A -85,B 0,C 180,E1 19592.64,E2 19592.64} C_VEL
LIN {X 0,Y 446.77,Z 422.643,A -85,B 0,C 180,E1 19591.274,E2 19591.274} C_VEL
LIN {X 0,Y 451.748,Z 429.041,A -85,B 0,C 180,E1 19589.875,E2 19589.875} C_VEL
LIN {X 0,Y 458.95,Z 438.496,A -85,B 0,C 180,E1 19587.997,E2 19587.997} C_VEL
LIN {X 0,Y 468.414,Z 451.673,A -85,B 0,C 180,E1 19585.736,E2 19585.736} C_VEL
LIN {X 0,Y 479.358,Z 467.882,A -85,B 0,C 180,E1 19583.357,E2 19583.357} C_VEL
LIN {X 0,Y 487.422,Z 480.855,A -85,B 0,C 180,E1 19581.728,E2 19581.728} C_VEL
LIN {X 0,Y 474.312,Z 734.538,A -85,B 0,C 180,E1 19577.744,E2 19577.744} C_VEL
LIN {X 0,Y 472.532,Z 757.416,A -85,B 0,C 180,E1 19577.301,E2 19577.301} C_VEL
LIN {X 0,Y 469.826,Z 781.616,A -85,B 0,C 180,E1 19576.667,E2 19576.667} C_VEL
LIN {X 0,Y 466.49,Z 803.749,A -85,B 0,C 180,E1 19575.894,E2 19575.894} C_VEL
LIN {X 0,Y 462.682,Z 825.268,A -85,B 0,C 180,E1 19574.965,E2 19574.965} C_VEL
LIN {X 0,Y 457.838,Z 848.459,A -85,B 0,C 180,E1 19573.726,E2 19573.726} C_VEL
LIN {X 0,Y 453.361,Z 867.266,A -85,B 0,C 180,E1 19572.531,E2 19572.531} C_VEL
LIN {X 0,Y 447.651,Z 889.182,A -85,B 0,C 180,E1 19570.878,E2 19570.878} C_VEL
LIN {X 0,Y 442.417,Z 907.348,A -85,B 0,C 180,E1 19569.258,E2 19569.258} C_VEL
LIN {X 0,Y 436.621,Z 926.505,A -85,B 0,C 180,E1 19567.281,E2 19567.281} C_VEL
LIN {X 0,Y 430.734,Z 944.563,A -85,B 0,C 180,E1 19565.067,E2 19565.067} C_VEL
LIN {X 0,Y 425.023,Z 961.78,A -85,B 0,C 180,E1 19562.625,E2 19562.625} C_VEL
LIN {X 0,Y 419.749,Z 977.254,A -85,B 0,C 180,E1 19560.016,E2 19560.016} C_VEL
LIN {X 0,Y 415.005,Z 991.499,A -85,B 0,C 180,E1 19557.244,E2 19557.244} C_VEL
LIN {X 0,Y 410.81,Z 1004.252,A -85,B 0,C 180,E1 19554.289,E2 19554.289} C_VEL
LIN {X 0,Y 407.422,Z 1015.332,A -85,B 0,C 180,E1 19551.298,E2 19551.298} C_VEL
LIN {X 0,Y 404.585,Z 1025.491,A -85,B 0,C 180,E1 19547.994,E2 19547.994} C_VEL
LIN {X 0,Y 402.711,Z 1033.254,A -85,B 0,C 180,E1 19544.964,E2 19544.964} C_VEL
LIN {X 0,Y 401.241,Z 1040.688,A -85,B 0,C 180,E1 19541.354,E2 19541.354} C_VEL
LIN {X 0,Y 400.515,Z 1045.483,A -85,B 0,C 180,E1 19538.326,E2 19538.326} C_VEL
LIN {X 0,Y 400.13,Z 1049.406,A -85,B 0,C 180,E1 19535.018,E2 19535.018} C_VEL
LIN {X 0,Y 399.993,Z 1051.738,A -85,B 0,C 180,E1 19531.719,E2 19531.719} C_VEL
LIN {X 0,Y 399.963,Z 1052.647,A -85,B 0,C 180,E1 19528.997,E2 19528.997} C_VEL
LIN {X 0,Y 399.966,Z 1052.589,A -85,B 0,C 180,E1 19526.13,E2 19526.13} C_VEL
LIN {X 0,Y 400.05,Z 1051.129,A -85,B 0,C 180,E1 19522.677,E2 19522.677} C_VEL
LIN {X 0,Y 400.254,Z 1048.492,A -85,B 0,C 180,E1 19519.638,E2 19519.638} C_VEL
LIN {X 0,Y 400.372,Z 1047.462,A -85,B 0,C 180,E1 19518.682,E2 19518.682} C_VEL
LIN {X 0,Y 399.552,Z 1046.226,A -85,B 0,C 180,E1 19517.591,E2 19517.591} C_VEL
LIN {X 0,Y 393.933,Z 1042.172,A -85,B 0,C 180,E1 19514.599,E2 19514.599} C_VEL
LIN {X 0,Y 393.592,Z 1040.768,A -85,B 0,C 180,E1 19513.731,E2 19513.731} C_VEL
LIN {X 0,Y 395.335,Z 1033.293,A -85,B 0,C 180,E1 19510.035,E2 19510.035} C_VEL
LIN {X 0,Y 397.439,Z 1025.806,A -85,B 0,C 180,E1 19507.043,E2 19507.043} C_VEL
LIN {X 0,Y 400.862,Z 1015.037,A -85,B 0,C 180,E1 19503.481,E2 19503.481} C_VEL
LIN {X 0,Y 404.547,Z 1004.329,A -85,B 0,C 180,E1 19500.537,E2 19500.537} C_VEL
LIN {X 0,Y 409.456,Z 990.937,A -85,B 0,C 180,E1 19497.404,E2 19497.404} C_VEL
LIN {X 0,Y 414.371,Z 977.647,A -85,B 0,C 180,E1 19494.78,E2 19494.78} C_VEL
LIN {X 0,Y 420.216,Z 962.118,A -85,B 0,C 180,E1 19492.128,E2 19492.128} C_VEL
LIN {X 0,Y 426.245,Z 945.497,A -85,B 0,C 180,E1 19489.739,E2 19489.739} C_VEL
LIN {X 0,Y 432.123,Z 928.921,A -85,B 0,C 180,E1 19487.674,E2 19487.674} C_VEL
LIN {X 0,Y 438.674,Z 909.227,A -85,B 0,C 180,E1 19485.592,E2 19485.592} C_VEL
LIN {X 0,Y 444.103,Z 891.864,A -85,B 0,C 180,E1 19484.022,E2 19484.022} C_VEL
LIN {X 0,Y 450.388,Z 869.901,A -85,B 0,C 180,E1 19482.33,E2 19482.33} C_VEL
LIN {X 0,Y 455.489,Z 850.06,A -85,B 0,C 180,E1 19481.057,E2 19481.057} C_VEL
LIN {X 0,Y 460.518,Z 828.114,A -85,B 0,C 180,E1 19479.867,E2 19479.867} C_VEL
LIN {X 0,Y 464.9,Z 805.136,A -85,B 0,C 180,E1 19478.87,E2 19478.87} C_VEL
LIN {X 0,Y 468.531,Z 782.725,A -85,B 0,C 180,E1 19478.087,E2 19478.087} C_VEL
LIN {X 0,Y 471.493,Z 758.275,A -85,B 0,C 180,E1 19477.445,E2 19477.445} C_VEL
LIN {X 0,Y 473.398,Z 735.671,A -85,B 0,C 180,E1 19477.007,E2 19477.007} C_VEL
LIN {X 0,Y 487.324,Z 487.631,A -85,B 0,C 180,E1 19473.096,E2 19473.096} C_VEL
LIN {X 0,Y 476.642,Z 471.149,A -85,B 0,C 180,E1 19470.683,E2 19470.683} C_VEL
LIN {X 0,Y 468.164,Z 458.897,A -85,B 0,C 180,E1 19468.582,E2 19468.582} C_VEL
LIN {X 0,Y 460.095,Z 447.835,A -85,B 0,C 180,E1 19466.387,E2 19466.387} C_VEL
LIN {X 0,Y 453.331,Z 438.974,A -85,B 0,C 180,E1 19464.359,E2 19464.359} C_VEL
LIN {X 0,Y 449.328,Z 433.847,A -85,B 0,C 180,E1 19463.058,E2 19463.058} C_VEL
LIN {X 0,Y 445.527,Z 429.019,A -85,B 0,C 180,E1 19461.735,E2 19461.735} C_VEL
LIN {X 0,Y 441.138,Z 423.591,A -85,B 0,C 180,E1 19460.084,E2 19460.084} C_VEL
LIN {X 0,Y 437.433,Z 419.055,A -85,B 0,C 180,E1 19458.56,E2 19458.56} C_VEL
LIN {X 0,Y 432.902,Z 413.914,A -85,B 0,C 180,E1 19456.505,E2 19456.505} C_VEL
LIN {X 0,Y 431.916,Z 412.287,A -85,B 0,C 180,E1 19455.991,E2 19455.991} C_VEL
LIN {X 0,Y 428.332,Z 408.967,A -85,B 0,C 180,E1 19454.119,E2 19454.119} C_VEL
LIN {X 0,Y 426.568,Z 406.004,A -85,B 0,C 180,E1 19453.005,E2 19453.005} C_VEL
LIN {X 0,Y 423.227,Z 403.422,A -85,B 0,C 180,E1 19450.826,E2 19450.826} C_VEL
LIN {X 0,Y 421.302,Z 399.897,A -85,B 0,C 180,E1 19449.15,E2 19449.15} C_VEL
LIN {X 0,Y 416.05,Z 394.962,A -85,B 0,C 180,E1 19442.066,E2 19442.066} C_VEL
LIN {X 0,Y 415.69,Z 393.552,A -85,B 0,C 180,E1 19439.311,E2 19439.311} C_VEL
LIN {X 0,Y 415.834,Z 394.29,A -85,B 0,C 180,E1 19437.244,E2 19437.244} C_VEL
LIN {X 0,Y 420.213,Z 399.241,A -85,B 0,C 180,E1 19430.135,E2 19430.135} C_VEL
LIN {X 0,Y 421.299,Z 399.833,A -85,B 0,C 180,E1 19429.193,E2 19429.193} C_VEL
LIN {X 0,Y 423.392,Z 403.66,A -85,B 0,C 180,E1 19427.382,E2 19427.382} C_VEL
LIN {X 0,Y 426.925,Z 406.472,A -85,B 0,C 180,E1 19425.105,E2 19425.105} C_VEL
LIN {X 0,Y 429.477,Z 410.381,A -85,B 0,C 180,E1 19423.568,E2 19423.568} C_VEL
LIN {X 0,Y 432.221,Z 412.744,A -85,B 0,C 180,E1 19422.185,E2 19422.185} C_VEL
LIN {X 0,Y 435.466,Z 417.05,A -85,B 0,C 180,E1 19420.622,E2 19420.622} C_VEL
LIN {X 0,Y 437.511,Z 419.106,A -85,B 0,C 180,E1 19419.742,E2 19419.742} C_VEL
LIN {X 0,Y 441.143,Z 423.609,A -85,B 0,C 180,E1 19418.248,E2 19418.248} C_VEL
LIN {X 0,Y 448.143,Z 432.936,A -85,B 0,C 180,E1 19415.656,E2 19415.656} C_VEL
LIN {X 0,Y 457.39,Z 446.075,A -85,B 0,C 180,E1 19412.672,E2 19412.672} C_VEL
LIN {X 0,Y 467.572,Z 461.659,A -85,B 0,C 180,E1 19409.796,E2 19409.796} C_VEL
LIN {X 0,Y 476.832,Z 476.803,A -85,B 0,C 180,E1 19407.455,E2 19407.455} C_VEL
LIN {X 0,Y 486.373,Z 493.527,A -85,B 0,C 180,E1 19405.251,E2 19405.251} C_VEL
LIN {X 0,Y 487.083,Z 495.289,A -85,B 0,C 180,E1 19405.083,E2 19405.083} C_VEL
LIN {X 0,Y 473.174,Z 745.34,A -85,B 0,C 180,E1 19401.141,E2 19401.141} C_VEL
LIN {X 0,Y 471.117,Z 771.554,A -85,B 0,C 180,E1 19400.661,E2 19400.661} C_VEL
LIN {X 0,Y 468.45,Z 793.432,A -85,B 0,C 180,E1 19400.133,E2 19400.133} C_VEL
LIN {X 0,Y 464.436,Z 818.378,A -85,B 0,C 180,E1 19399.334,E2 19399.334} C_VEL
LIN {X 0,Y 460.667,Z 837.803,A -85,B 0,C 180,E1 19398.546,E2 19398.546} C_VEL
LIN {X 0,Y 455.615,Z 860.692,A -85,B 0,C 180,E1 19397.416,E2 19397.416} C_VEL
LIN {X 0,Y 450.208,Z 881.742,A -85,B 0,C 180,E1 19396.137,E2 19396.137} C_VEL
LIN {X 0,Y 444.695,Z 901.411,A -85,B 0,C 180,E1 19394.731,E2 19394.731} C_VEL
LIN {X 0,Y 438.111,Z 922.871,A -85,B 0,C 180,E1 19392.894,E2 19392.894} C_VEL
LIN {X 0,Y 432.585,Z 939.743,A -85,B 0,C 180,E1 19391.205,E2 19391.205} C_VEL
LIN {X 0,Y 425.755,Z 959.582,A -85,B 0,C 180,E1 19388.882,E2 19388.882} C_VEL
LIN {X 0,Y 420.065,Z 975.509,A -85,B 0,C 180,E1 19386.688,E2 19386.688} C_VEL
LIN {X 0,Y 414.175,Z 991.959,A -85,B 0,C 180,E1 19384.062,E2 19384.062} C_VEL
LIN {X 0,Y 409.032,Z 1006.203,A -85,B 0,C 180,E1 19381.378,E2 19381.378} C_VEL
LIN {X 0,Y 404.256,Z 1020.075,A -85,B 0,C 180,E1 19378.352,E2 19378.352} C_VEL
LIN {X 0,Y 400.198,Z 1032.366,A -85,B 0,C 180,E1 19375.134,E2 19375.134} C_VEL
LIN {X 0,Y 396.98,Z 1043.425,A -85,B 0,C 180,E1 19371.731,E2 19371.731} C_VEL
LIN {X 0,Y 394.684,Z 1052.453,A -85,B 0,C 180,E1 19368.309,E2 19368.309} C_VEL
LIN {X 0,Y 393.201,Z 1059.93,A -85,B 0,C 180,E1 19364.883,E2 19364.883} C_VEL
LIN {X 0,Y 392.369,Z 1065.631,A -85,B 0,C 180,E1 19361.465,E2 19361.465} C_VEL
LIN {X 0,Y 392.048,Z 1069.387,A -85,B 0,C 180,E1 19358.507,E2 19358.507} C_VEL
LIN {X 0,Y 391.95,Z 1072.381,A -85,B 0,C 180,E1 19355.123,E2 19355.123} C_VEL
LIN {X 0,Y 391.951,Z 1073.728,A -85,B 0,C 180,E1 19351.754,E2 19351.754} C_VEL
LIN {X 0,Y 391.962,Z 1073.786,A -85,B 0,C 180,E1 19348.977,E2 19348.977} C_VEL
LIN {X 0,Y 391.946,Z 1072.78,A -85,B 0,C 180,E1 19346.05,E2 19346.05} C_VEL
LIN {X 0,Y 391.991,Z 1070.094,A -85,B 0,C 180,E1 19342.525,E2 19342.525} C_VEL
LIN {X 0,Y 392.226,Z 1066.319,A -85,B 0,C 180,E1 19339.424,E2 19339.424} C_VEL
LIN {X 0,Y 392.778,Z 1061.56,A -85,B 0,C 180,E1 19336.455,E2 19336.455} C_VEL
LIN {X 0,Y 394.093,Z 1053.874,A -85,B 0,C 180,E1 19332.731,E2 19332.731} C_VEL
LIN {X 0,Y 395.874,Z 1045.813,A -85,B 0,C 180,E1 19329.601,E2 19329.601} C_VEL
LIN {X 0,Y 398.671,Z 1035.288,A -85,B 0,C 180,E1 19326.184,E2 19326.184} C_VEL
LIN {X 0,Y 401.884,Z 1024.381,A -85,B 0,C 180,E1 19323.235,E2 19323.235} C_VEL
LIN {X 0,Y 406.125,Z 1011.269,A -85,B 0,C 180,E1 19320.177,E2 19320.177} C_VEL
LIN {X 0,Y 410.98,Z 996.617,A -85,B 0,C 180,E1 19317.309,E2 19317.309} C_VEL
LIN {X 0,Y 416.102,Z 981.703,A -85,B 0,C 180,E1 19314.78,E2 19314.78} C_VEL
LIN {X 0,Y 422.052,Z 964.053,A -85,B 0,C 180,E1 19312.236,E2 19312.236} C_VEL
LIN {X 0,Y 427.606,Z 947.296,A -85,B 0,C 180,E1 19310.156,E2 19310.156} C_VEL
LIN {X 0,Y 434.076,Z 926.837,A -85,B 0,C 180,E1 19307.997,E2 19307.997} C_VEL
LIN {X 0,Y 439.355,Z 909.137,A -85,B 0,C 180,E1 19306.404,E2 19306.404} C_VEL
LIN {X 0,Y 445.485,Z 887.007,A -85,B 0,C 180,E1 19304.709,E2 19304.709} C_VEL
LIN {X 0,Y 450.401,Z 867.335,A -85,B 0,C 180,E1 19303.453,E2 19303.453} C_VEL
